KUKA KRL program: EPS_2_26056_SANMH1A_A_20260107125654.src

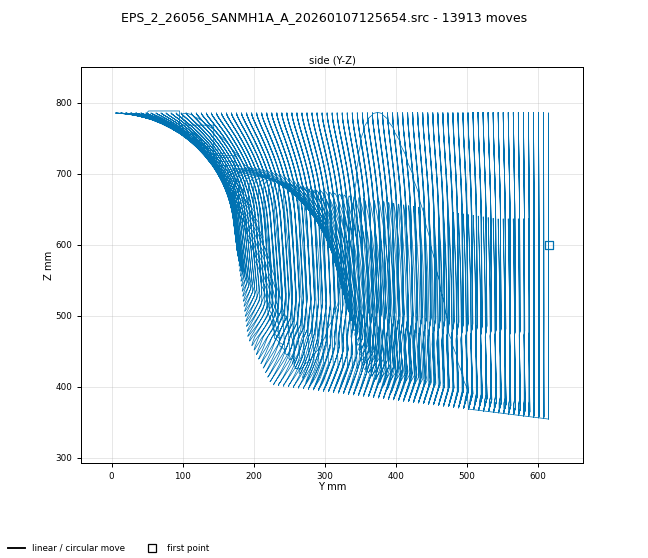
[picture p0: tool path of EPS_2_26056_SANMH1A_A_20260107125654.src, 13913 of 13915 moves have a stored position in this frame; points joined in program order, loops and branches not executed]
&ACCESS RVP
&REL 4
&COMMENT QRS 19112012
&PARAM EDITMASK = *
DEF PART()
EXT BAS (BAS_COMMAND :IN,REAL :IN )
INT I
BAS (#INITMOV,0 )

;KUKA QRS Post kuka4.cps  Date:22-06-2017 !

File_ID=2959

QRS_PRE_INIT()

;Init var - Until changes are made in qrs_pre_init
Outlet_Square_prg=0
Inlet_1_Square_prg=0
Inlet_2_Square_prg=0
Inlet_3_Square_prg=0
Inlet_4_Square_prg=0
Inlet_5_Square_prg=0

Outlet_1={X 0.000, Y 512.360, Z 637.000, B 0.000, E1 0.000 }
Inlet_1={X 0.000, Y 512.360, Z 637.000, B 0.000, E1 180.000 }
Inlet_2={X 0.000, Y 540.930, Z 321.000, B 0.000, E1 270.000 }
Outlet_1_type=299
Inlet_1_type=299
Inlet_2_type=251
;QRS#1=Sidecore dimensions
;QRS#2=300-12" PVC SDR 35
;QRS#3=300-12" PVC SDR 35
;QRS#4=250-10" PVC SDR 35
;QRS#5=
;QRS#6=
;QRS#7=
;QRS#8=
;QRS#9=16M PSX
;QRS#10=16M PSX
;QRS#11=14M PSX
;QRS#12=
;QRS#13=
;QRS#14=
;QRS#15=
;QRS#16=1220x127x1067 3,5'
;QRS#17=EPS Height
;QRS#18=786,5
;QRS#19=*
;QRS#20= UPDATED VERSION 22-06-2017
;QRS#21=*
Outlet_Square=0150
Inlet_1_Square=0150
Inlet_2_Square=0100
Inlet_3_Square=0
Inlet_4_Square=0
Inlet_5_Square=0
Mill_Square=1
Outlet_Square_Prg=206
Inlet_1_Square_prg=206
Inlet_2_Square_prg=205

QRS_INIT()

$ADVANCE=5

; T1
PTP {E1 173.596,E2 173.596}
PTP {X 0,Y 615.515,A -85,B 0,C 180,E1 173.596,E2 173.596,E3 0,E4 0,E5 0,E6 0}
QRS_SPEED_INIT()
LIN {X 0,Y 615.515,Z 600,A -85,B 0,C 180,E1 173.596,E2 173.596,E3 0,E4 0,E5 0,E6 0} C_VEL
LIN {X 0,Y 615.515,Z 364.495,A -85,B 0,C 180,E1 173.596,E2 173.596} C_VEL
LIN {X 0,Y 615.515,Z 356.328,A -85,B 0,C 180,E1 173.596,E2 173.596} C_VEL
LIN {X 0,Y 615.484,Z 354.328,A -85,B 0,C 180,E1 173.41,E2 173.41} C_VEL
LIN {X 0,Y 615.426,Z 354.324,A -85,B 0,C 180,E1 170.8,E2 170.8} C_VEL
LIN {X 0,Y 615.427,Z 354.324,A -85,B 0,C 180,E1 168.806,E2 168.806} C_VEL
LIN {X 0,Y 615.427,Z 354.324,A -85,B 0,C 180,E1 166.797,E2 166.797} C_VEL
LIN {X 0,Y 615.426,Z 354.324,A -85,B 0,C 180,E1 164.772,E2 164.772} C_VEL
LIN {X 0,Y 615.424,Z 354.324,A -85,B 0,C 180,E1 162.728,E2 162.728} C_VEL
LIN {X 0,Y 615.42,Z 354.324,A -85,B 0,C 180,E1 160.66,E2 160.66} C_VEL
LIN {X 0,Y 615.416,Z 354.324,A -85,B 0,C 180,E1 158.565,E2 158.565} C_VEL
LIN {X 0,Y 615.413,Z 354.324,A -85,B 0,C 180,E1 156.441,E2 156.441} C_VEL
LIN {X 0,Y 615.412,Z 354.324,A -85,B 0,C 180,E1 154.281,E2 154.281} C_VEL
LIN {X 0,Y 615.465,Z 354.323,A -85,B 0,C 180,E1 151.55,E2 151.55} C_VEL
LIN {X 0,Y 615.448,Z 354.325,A -85,B 0,C 180,E1 148.917,E2 148.917} C_VEL
LIN {X 0,Y 615.415,Z 354.324,A -85,B 0,C 180,E1 146.473,E2 146.473} C_VEL
LIN {X 0,Y 615.412,Z 354.324,A -85,B 0,C 180,E1 144.173,E2 144.173} C_VEL
LIN {X 0,Y 615.422,Z 354.323,A -85,B 0,C 180,E1 141.927,E2 141.927} C_VEL
LIN {X 0,Y 615.467,Z 354.326,A -85,B 0,C 180,E1 139.392,E2 139.392} C_VEL
LIN {X 0,Y 615.436,Z 354.325,A -85,B 0,C 180,E1 136.751,E2 136.751} C_VEL
LIN {X 0,Y 615.411,Z 354.324,A -85,B 0,C 180,E1 134.154,E2 134.154} C_VEL
LIN {X 0,Y 615.413,Z 354.324,A -85,B 0,C 180,E1 132.072,E2 132.072} C_VEL
LIN {X 0,Y 615.43,Z 354.323,A -85,B 0,C 180,E1 129.753,E2 129.753} C_VEL
LIN {X 0,Y 615.465,Z 354.325,A -85,B 0,C 180,E1 126.934,E2 126.934} C_VEL
LIN {X 0,Y 615.413,Z 354.324,A -85,B 0,C 180,E1 124.025,E2 124.025} C_VEL
LIN {X 0,Y 615.431,Z 354.323,A -85,B 0,C 180,E1 121.687,E2 121.687} C_VEL
LIN {X 0,Y 615.498,Z 354.495,A -85,B 0,C 180,E1 118.983,E2 118.983} C_VEL
LIN {X 0,Y 615.499,Z 355.379,A -85,B 0,C 180,E1 118.842,E2 118.842} C_VEL
LIN {X 0,Y 615.468,Z 383.107,A -85,B 0,C 180,E1 116.261,E2 116.261} C_VEL
LIN {X 0,Y 615.463,Z 411.593,A -85,B 0,C 180,E1 113.667,E2 113.667} C_VEL
LIN {X 0,Y 615.498,Z 440.574,A -85,B 0,C 180,E1 111.079,E2 111.079} C_VEL
LIN {X 0,Y 615.486,Z 472.602,A -85,B 0,C 180,E1 108.278,E2 108.278} C_VEL
LIN {X 0,Y 615.487,Z 474.74,A -85,B 0,C 180,E1 108.197,E2 108.197} C_VEL
LIN {X 0,Y 615.498,Z 640.194,A -85,B 0,C 180,E1 106.201,E2 106.201} C_VEL
LIN {X 0,Y 615.49,Z 654.874,A -85,B 0,C 180,E1 105.904,E2 105.904} C_VEL
LIN {X 0,Y 615.48,Z 669.457,A -85,B 0,C 180,E1 105.479,E2 105.479} C_VEL
LIN {X 0,Y 615.492,Z 682.768,A -85,B 0,C 180,E1 104.971,E2 104.971} C_VEL
LIN {X 0,Y 615.485,Z 696.395,A -85,B 0,C 180,E1 104.319,E2 104.319} C_VEL
LIN {X 0,Y 615.5,Z 709.685,A -85,B 0,C 180,E1 103.536,E2 103.536} C_VEL
LIN {X 0,Y 615.497,Z 721.532,A -85,B 0,C 180,E1 102.696,E2 102.696} C_VEL
LIN {X 0,Y 615.497,Z 733.373,A -85,B 0,C 180,E1 101.692,E2 101.692} C_VEL
LIN {X 0,Y 615.495,Z 743.166,A -85,B 0,C 180,E1 100.708,E2 100.708} C_VEL
LIN {X 0,Y 615.495,Z 753.021,A -85,B 0,C 180,E1 99.529,E2 99.529} C_VEL
LIN {X 0,Y 615.497,Z 761.11,A -85,B 0,C 180,E1 98.37,E2 98.37} C_VEL
LIN {X 0,Y 615.492,Z 767.789,A -85,B 0,C 180,E1 97.214,E2 97.214} C_VEL
LIN {X 0,Y 615.495,Z 773.954,A -85,B 0,C 180,E1 95.897,E2 95.897} C_VEL
LIN {X 0,Y 615.489,Z 778.72,A -85,B 0,C 180,E1 94.583,E2 94.583} C_VEL
LIN {X 0,Y 615.491,Z 782.223,A -85,B 0,C 180,E1 93.272,E2 93.272} C_VEL
LIN {X 0,Y 615.499,Z 784.541,A -85,B 0,C 180,E1 91.962,E2 91.962} C_VEL
LIN {X 0,Y 615.491,Z 785.728,A -85,B 0,C 180,E1 90.653,E2 90.653} C_VEL
LIN {X 0,Y 615.492,Z 785.751,A -85,B 0,C 180,E1 89.345,E2 89.345} C_VEL
LIN {X 0,Y 615.499,Z 784.644,A -85,B 0,C 180,E1 88.036,E2 88.036} C_VEL
LIN {X 0,Y 615.494,Z 782.413,A -85,B 0,C 180,E1 86.726,E2 86.726} C_VEL
LIN {X 0,Y 615.49,Z 779.002,A -85,B 0,C 180,E1 85.415,E2 85.415} C_VEL
LIN {X 0,Y 615.496,Z 774.332,A -85,B 0,C 180,E1 84.101,E2 84.101} C_VEL
LIN {X 0,Y 615.494,Z 768.266,A -85,B 0,C 180,E1 82.783,E2 82.783} C_VEL
LIN {X 0,Y 615.49,Z 760.627,A -85,B 0,C 180,E1 81.462,E2 81.462} C_VEL
LIN {X 0,Y 615.496,Z 752.443,A -85,B 0,C 180,E1 80.303,E2 80.303} C_VEL
LIN {X 0,Y 615.496,Z 742.329,A -85,B 0,C 180,E1 79.108,E2 79.108} C_VEL
LIN {X 0,Y 615.498,Z 730.672,A -85,B 0,C 180,E1 77.971,E2 77.971} C_VEL
LIN {X 0,Y 615.498,Z 719.4,A -85,B 0,C 180,E1 77.05,E2 77.05} C_VEL
LIN {X 0,Y 615.498,Z 707.158,A -85,B 0,C 180,E1 76.209,E2 76.209} C_VEL
LIN {X 0,Y 615.478,Z 693.757,A -85,B 0,C 180,E1 75.45,E2 75.45} C_VEL
LIN {X 0,Y 615.492,Z 679.889,A -85,B 0,C 180,E1 74.816,E2 74.816} C_VEL
LIN {X 0,Y 615.481,Z 665.667,A -85,B 0,C 180,E1 74.306,E2 74.306} C_VEL
LIN {X 0,Y 615.499,Z 651.574,A -85,B 0,C 180,E1 73.93,E2 73.93} C_VEL
LIN {X 0,Y 615.497,Z 637.157,A -85,B 0,C 180,E1 73.666,E2 73.666} C_VEL
LIN {X 0,Y 615.484,Z 473.34,A -85,B 0,C 180,E1 71.681,E2 71.681} C_VEL
LIN {X 0,Y 615.494,Z 445.533,A -85,B 0,C 180,E1 69.269,E2 69.269} C_VEL
LIN {X 0,Y 615.495,Z 415.789,A -85,B 0,C 180,E1 66.622,E2 66.622} C_VEL
LIN {X 0,Y 615.489,Z 386.043,A -85,B 0,C 180,E1 63.92,E2 63.92} C_VEL
LIN {X 0,Y 615.497,Z 356.297,A -85,B 0,C 180,E1 61.155,E2 61.155} C_VEL
LIN {X 0,Y 615.497,Z 354.615,A -85,B 0,C 180,E1 60.968,E2 60.968} C_VEL
LIN {X 0,Y 615.425,Z 354.325,A -85,B 0,C 180,E1 60.216,E2 60.216} C_VEL
LIN {X 0,Y 615.432,Z 354.325,A -85,B 0,C 180,E1 58.311,E2 58.311} C_VEL
LIN {X 0,Y 615.41,Z 354.325,A -85,B 0,C 180,E1 55.972,E2 55.972} C_VEL
LIN {X 0,Y 615.46,Z 354.325,A -85,B 0,C 180,E1 53.067,E2 53.067} C_VEL
LIN {X 0,Y 615.429,Z 354.324,A -85,B 0,C 180,E1 50.245,E2 50.245} C_VEL
LIN {X 0,Y 615.414,Z 354.324,A -85,B 0,C 180,E1 47.928,E2 47.928} C_VEL
LIN {X 0,Y 615.413,Z 354.324,A -85,B 0,C 180,E1 45.843,E2 45.843} C_VEL
LIN {X 0,Y 615.442,Z 354.324,A -85,B 0,C 180,E1 43.249,E2 43.249} C_VEL
LIN {X 0,Y 615.47,Z 354.323,A -85,B 0,C 180,E1 40.608,E2 40.608} C_VEL
LIN {X 0,Y 615.423,Z 354.322,A -85,B 0,C 180,E1 38.004,E2 38.004} C_VEL
LIN {X 0,Y 615.422,Z 354.323,A -85,B 0,C 180,E1 35.62,E2 35.62} C_VEL
LIN {X 0,Y 615.448,Z 354.324,A -85,B 0,C 180,E1 33.239,E2 33.239} C_VEL
LIN {X 0,Y 615.489,Z 354.325,A -85,B 0,C 180,E1 30.92,E2 30.92} C_VEL
LIN {X 0,Y 615.468,Z 354.319,A -85,B 0,C 180,E1 28.446,E2 28.446} C_VEL
LIN {X 0,Y 615.468,Z 354.318,A -85,B 0,C 180,E1 26.445,E2 26.445} C_VEL
LIN {X 0,Y 615.433,Z 354.32,A -85,B 0,C 180,E1 23.996,E2 23.996} C_VEL
LIN {X 0,Y 615.443,Z 354.319,A -85,B 0,C 180,E1 22.138,E2 22.138} C_VEL
LIN {X 0,Y 615.437,Z 354.319,A -85,B 0,C 180,E1 20.035,E2 20.035} C_VEL
LIN {X 0,Y 615.498,Z 354.519,A -85,B 0,C 180,E1 18.797,E2 18.797} C_VEL
LIN {X 0,Y 615.492,Z 371.153,A -85,B 0,C 180,E1 16.167,E2 16.167} C_VEL
LIN {X 0,Y 615.457,Z 375.25,A -85,B 0,C 180,E1 15.566,E2 15.566} C_VEL
LIN {X 0,Y 615.454,Z 377.392,A -85,B 0,C 180,E1 15.503,E2 15.503} C_VEL
LIN {X 0,Y 615.498,Z 511.173,A -85,B 0,C 180,E1 13.905,E2 13.905} C_VEL
LIN {X 0,Y 615.497,Z 524.744,A -85,B 0,C 180,E1 13.621,E2 13.621} C_VEL
LIN {X 0,Y 615.497,Z 538.485,A -85,B 0,C 180,E1 13.201,E2 13.201} C_VEL
LIN {X 0,Y 615.493,Z 550.898,A -85,B 0,C 180,E1 12.698,E2 12.698} C_VEL
LIN {X 0,Y 615.486,Z 563.841,A -85,B 0,C 180,E1 12.028,E2 12.028} C_VEL
LIN {X 0,Y 615.499,Z 575.557,A -85,B 0,C 180,E1 11.276,E2 11.276} C_VEL
LIN {X 0,Y 615.498,Z 587.225,A -85,B 0,C 180,E1 10.36,E2 10.36} C_VEL
LIN {X 0,Y 615.497,Z 597.649,A -85,B 0,C 180,E1 9.364,E2 9.364} C_VEL
LIN {X 0,Y 615.496,Z 606.239,A -85,B 0,C 180,E1 8.371,E2 8.371} C_VEL
LIN {X 0,Y 615.495,Z 614.452,A -85,B 0,C 180,E1 7.216,E2 7.216} C_VEL
LIN {X 0,Y 615.496,Z 620.183,A -85,B 0,C 180,E1 6.227,E2 6.227} C_VEL
LIN {X 0,Y 615.495,Z 624.887,A -85,B 0,C 180,E1 5.241,E2 5.241} C_VEL
LIN {X 0,Y 615.494,Z 629.757,A -85,B 0,C 180,E1 3.929,E2 3.929} C_VEL
LIN {X 0,Y 615.496,Z 633.154,A -85,B 0,C 180,E1 2.618,E2 2.618} C_VEL
LIN {X 0,Y 615.494,Z 635.174,A -85,B 0,C 180,E1 1.309,E2 1.309} C_VEL
LIN {X 0,Y 615.491,Z 635.885,A -85,B 0,C 180,E1 0,E2 0} C_VEL
LIN {X 0,Y 615.489,Z 635.28,A -85,B 0,C 180,E1 -1.309,E2 -1.309} C_VEL
LIN {X 0,Y 615.497,Z 633.35,A -85,B 0,C 180,E1 -2.618,E2 -2.618} C_VEL
LIN {X 0,Y 615.494,Z 630.046,A -85,B 0,C 180,E1 -3.928,E2 -3.928} C_VEL
LIN {X 0,Y 615.495,Z 625.274,A -85,B 0,C 180,E1 -5.241,E2 -5.241} C_VEL
LIN {X 0,Y 615.497,Z 618.874,A -85,B 0,C 180,E1 -6.557,E2 -6.557} C_VEL
LIN {X 0,Y 615.496,Z 611.744,A -85,B 0,C 180,E1 -7.71,E2 -7.71} C_VEL
LIN {X 0,Y 615.498,Z 604.271,A -85,B 0,C 180,E1 -8.702,E2 -8.702} C_VEL
LIN {X 0,Y 615.495,Z 595.292,A -85,B 0,C 180,E1 -9.696,E2 -9.696} C_VEL
LIN {X 0,Y 615.498,Z 584.208,A -85,B 0,C 180,E1 -10.709,E2 -10.709} C_VEL
LIN {X 0,Y 615.498,Z 573.281,A -85,B 0,C 180,E1 -11.526,E2 -11.526} C_VEL
LIN {X 0,Y 615.486,Z 560.984,A -85,B 0,C 180,E1 -12.279,E2 -12.279} C_VEL
LIN {X 0,Y 615.488,Z 549.146,A -85,B 0,C 180,E1 -12.865,E2 -12.865} C_VEL
LIN {X 0,Y 615.494,Z 536.22,A -85,B 0,C 180,E1 -13.369,E2 -13.369} C_VEL
LIN {X 0,Y 615.498,Z 523.24,A -85,B 0,C 180,E1 -13.748,E2 -13.748} C_VEL
LIN {X 0,Y 615.497,Z 510.029,A -85,B 0,C 180,E1 -14.012,E2 -14.012} C_VEL
LIN {X 0,Y 615.491,Z 375.663,A -85,B 0,C 180,E1 -15.629,E2 -15.629} C_VEL
LIN {X 0,Y 615.495,Z 374.551,A -85,B 0,C 180,E1 -15.735,E2 -15.735} C_VEL
LIN {X 0,Y 615.496,Z 355.917,A -85,B 0,C 180,E1 -18.646,E2 -18.646} C_VEL
LIN {X 0,Y 615.496,Z 354.46,A -85,B 0,C 180,E1 -18.905,E2 -18.905} C_VEL
LIN {X 0,Y 615.491,Z 354.311,A -85,B 0,C 180,E1 -21.432,E2 -21.432} C_VEL
LIN {X 0,Y 615.469,Z 354.316,A -85,B 0,C 180,E1 -24.273,E2 -24.273} C_VEL
LIN {X 0,Y 615.481,Z 354.319,A -85,B 0,C 180,E1 -27.043,E2 -27.043} C_VEL
LIN {X 0,Y 615.488,Z 354.308,A -85,B 0,C 180,E1 -29.794,E2 -29.794} C_VEL
LIN {X 0,Y 615.487,Z 354.323,A -85,B 0,C 180,E1 -32.457,E2 -32.457} C_VEL
LIN {X 0,Y 615.476,Z 354.32,A -85,B 0,C 180,E1 -34.816,E2 -34.816} C_VEL
LIN {X 0,Y 615.467,Z 354.314,A -85,B 0,C 180,E1 -37.244,E2 -37.244} C_VEL
LIN {X 0,Y 615.489,Z 354.318,A -85,B 0,C 180,E1 -40.088,E2 -40.088} C_VEL
LIN {X 0,Y 615.494,Z 354.325,A -85,B 0,C 180,E1 -42.352,E2 -42.352} C_VEL
LIN {X 0,Y 615.448,Z 354.317,A -85,B 0,C 180,E1 -45.072,E2 -45.072} C_VEL
LIN {X 0,Y 615.497,Z 354.318,A -85,B 0,C 180,E1 -47.919,E2 -47.919} C_VEL
LIN {X 0,Y 615.475,Z 354.325,A -85,B 0,C 180,E1 -50.248,E2 -50.248} C_VEL
LIN {X 0,Y 615.43,Z 354.322,A -85,B 0,C 180,E1 -52.753,E2 -52.753} C_VEL
LIN {X 0,Y 615.438,Z 354.322,A -85,B 0,C 180,E1 -55.306,E2 -55.306} C_VEL
LIN {X 0,Y 615.438,Z 354.325,A -85,B 0,C 180,E1 -58.311,E2 -58.311} C_VEL
LIN {X 0,Y 615.416,Z 354.325,A -85,B 0,C 180,E1 -60.589,E2 -60.589} C_VEL
LIN {X 0,Y 615.496,Z 354.507,A -85,B 0,C 180,E1 -61.886,E2 -61.886} C_VEL
LIN {X 0,Y 615.494,Z 355.377,A -85,B 0,C 180,E1 -62.018,E2 -62.018} C_VEL
LIN {X 0,Y 615.482,Z 387.128,A -85,B 0,C 180,E1 -64.721,E2 -64.721} C_VEL
LIN {X 0,Y 615.499,Z 419.368,A -85,B 0,C 180,E1 -67.404,E2 -67.404} C_VEL
LIN {X 0,Y 615.479,Z 452.912,A -85,B 0,C 180,E1 -70.14,E2 -70.14} C_VEL
LIN {X 0,Y 615.486,Z 472.762,A -85,B 0,C 180,E1 -71.72,E2 -71.72} C_VEL
LIN {X 0,Y 615.498,Z 640.913,A -85,B 0,C 180,E1 -73.764,E2 -73.764} C_VEL
LIN {X 0,Y 615.49,Z 656.681,A -85,B 0,C 180,E1 -74.094,E2 -74.094} C_VEL
LIN {X 0,Y 615.48,Z 672.028,A -85,B 0,C 180,E1 -74.561,E2 -74.561} C_VEL
LIN {X 0,Y 615.484,Z 685.734,A -85,B 0,C 180,E1 -75.112,E2 -75.112} C_VEL
LIN {X 0,Y 615.493,Z 700.041,A -85,B 0,C 180,E1 -75.833,E2 -75.833} C_VEL
LIN {X 0,Y 615.497,Z 712.886,A -85,B 0,C 180,E1 -76.63,E2 -76.63} C_VEL
LIN {X 0,Y 615.495,Z 725.244,A -85,B 0,C 180,E1 -77.553,E2 -77.553} C_VEL
LIN {X 0,Y 615.495,Z 735.597,A -85,B 0,C 180,E1 -78.473,E2 -78.473} C_VEL
LIN {X 0,Y 615.494,Z 745.176,A -85,B 0,C 180,E1 -79.472,E2 -79.472} C_VEL
LIN {X 0,Y 615.495,Z 754.57,A -85,B 0,C 180,E1 -80.635,E2 -80.635} C_VEL
LIN {X 0,Y 615.496,Z 762.375,A -85,B 0,C 180,E1 -81.793,E2 -81.793} C_VEL
LIN {X 0,Y 615.497,Z 769.605,A -85,B 0,C 180,E1 -83.102,E2 -83.102} C_VEL
LIN {X 0,Y 615.499,Z 775.433,A -85,B 0,C 180,E1 -84.429,E2 -84.429} C_VEL
LIN {X 0,Y 615.491,Z 778.857,A -85,B 0,C 180,E1 -85.415,E2 -85.415} C_VEL
LIN {X 0,Y 615.492,Z 782.316,A -85,B 0,C 180,E1 -86.726,E2 -86.726} C_VEL
LIN {X 0,Y 615.496,Z 784.592,A -85,B 0,C 180,E1 -88.036,E2 -88.036} C_VEL
LIN {X 0,Y 615.493,Z 785.74,A -85,B 0,C 180,E1 -89.345,E2 -89.345} C_VEL
LIN {X 0,Y 615.493,Z 785.741,A -85,B 0,C 180,E1 -90.653,E2 -90.653} C_VEL
LIN {X 0,Y 615.495,Z 784.595,A -85,B 0,C 180,E1 -91.962,E2 -91.962} C_VEL
LIN {X 0,Y 615.492,Z 782.32,A -85,B 0,C 180,E1 -93.272,E2 -93.272} C_VEL
LIN {X 0,Y 615.491,Z 778.864,A -85,B 0,C 180,E1 -94.583,E2 -94.583} C_VEL
LIN {X 0,Y 615.49,Z 774.148,A -85,B 0,C 180,E1 -95.897,E2 -95.897} C_VEL
LIN {X 0,Y 615.496,Z 768.035,A -85,B 0,C 180,E1 -97.214,E2 -97.214} C_VEL
LIN {X 0,Y 615.49,Z 760.341,A -85,B 0,C 180,E1 -98.535,E2 -98.535} C_VEL
LIN {X 0,Y 615.495,Z 752.122,A -85,B 0,C 180,E1 -99.695,E2 -99.695} C_VEL
LIN {X 0,Y 615.496,Z 741.897,A -85,B 0,C 180,E1 -100.892,E2 -100.892} C_VEL
LIN {X 0,Y 615.495,Z 732.08,A -85,B 0,C 180,E1 -101.859,E2 -101.859} C_VEL
LIN {X 0,Y 615.497,Z 719.964,A -85,B 0,C 180,E1 -102.864,E2 -102.864} C_VEL
LIN {X 0,Y 615.498,Z 707.816,A -85,B 0,C 180,E1 -103.704,E2 -103.704} C_VEL
LIN {X 0,Y 615.477,Z 694.399,A -85,B 0,C 180,E1 -104.472,E2 -104.472} C_VEL
LIN {X 0,Y 615.495,Z 679.877,A -85,B 0,C 180,E1 -105.14,E2 -105.14} C_VEL
LIN {X 0,Y 615.48,Z 665.654,A -85,B 0,C 180,E1 -105.649,E2 -105.649} C_VEL
LIN {X 0,Y 615.5,Z 651.125,A -85,B 0,C 180,E1 -106.036,E2 -106.036} C_VEL
LIN {X 0,Y 615.498,Z 636.349,A -85,B 0,C 180,E1 -106.301,E2 -106.301} C_VEL
LIN {X 0,Y 615.487,Z 472.791,A -85,B 0,C 180,E1 -108.279,E2 -108.279} C_VEL
LIN {X 0,Y 615.481,Z 441.108,A -85,B 0,C 180,E1 -110.817,E2 -110.817} C_VEL
LIN {X 0,Y 615.487,Z 407.768,A -85,B 0,C 180,E1 -113.555,E2 -113.555} C_VEL
LIN {X 0,Y 615.496,Z 374.428,A -85,B 0,C 180,E1 -116.351,E2 -116.351} C_VEL
LIN {X 0,Y 615.495,Z 354.685,A -85,B 0,C 180,E1 -118.062,E2 -118.062} C_VEL
LIN {X 0,Y 615.464,Z 354.326,A -85,B 0,C 180,E1 -118.446,E2 -118.446} C_VEL
LIN {X 0,Y 615.422,Z 354.324,A -85,B 0,C 180,E1 -120.922,E2 -120.922} C_VEL
LIN {X 0,Y 615.414,Z 354.323,A -85,B 0,C 180,E1 -123.239,E2 -123.239} C_VEL
LIN {X 0,Y 615.447,Z 354.322,A -85,B 0,C 180,E1 -125.828,E2 -125.828} C_VEL
LIN {X 0,Y 615.477,Z 354.322,A -85,B 0,C 180,E1 -128.067,E2 -128.067} C_VEL
LIN {X 0,Y 615.455,Z 354.324,A -85,B 0,C 180,E1 -130.607,E2 -130.607} C_VEL
LIN {X 0,Y 615.419,Z 354.324,A -85,B 0,C 180,E1 -133.041,E2 -133.041} C_VEL
LIN {X 0,Y 615.418,Z 354.324,A -85,B 0,C 180,E1 -135.073,E2 -135.073} C_VEL
LIN {X 0,Y 615.421,Z 354.324,A -85,B 0,C 180,E1 -137.641,E2 -137.641} C_VEL
LIN {X 0,Y 615.496,Z 354.322,A -85,B 0,C 180,E1 -140.251,E2 -140.251} C_VEL
LIN {X 0,Y 615.42,Z 354.324,A -85,B 0,C 180,E1 -143.069,E2 -143.069} C_VEL
LIN {X 0,Y 615.411,Z 354.324,A -85,B 0,C 180,E1 -145.307,E2 -145.307} C_VEL
LIN {X 0,Y 615.416,Z 354.323,A -85,B 0,C 180,E1 -147.538,E2 -147.538} C_VEL
LIN {X 0,Y 615.476,Z 354.323,A -85,B 0,C 180,E1 -150.204,E2 -150.204} C_VEL
LIN {X 0,Y 615.429,Z 354.324,A -85,B 0,C 180,E1 -152.962,E2 -152.962} C_VEL
LIN {X 0,Y 615.428,Z 354.324,A -85,B 0,C 180,E1 -155.006,E2 -155.006} C_VEL
LIN {X 0,Y 615.419,Z 354.324,A -85,B 0,C 180,E1 -157.153,E2 -157.153} C_VEL
LIN {X 0,Y 615.413,Z 354.323,A -85,B 0,C 180,E1 -159.457,E2 -159.457} C_VEL
LIN {X 0,Y 615.448,Z 354.323,A -85,B 0,C 180,E1 -162.042,E2 -162.042} C_VEL
LIN {X 0,Y 615.456,Z 354.325,A -85,B 0,C 180,E1 -164.773,E2 -164.773} C_VEL
LIN {X 0,Y 615.413,Z 354.324,A -85,B 0,C 180,E1 -167.468,E2 -167.468} C_VEL
LIN {X 0,Y 615.45,Z 354.323,A -85,B 0,C 180,E1 -170.137,E2 -170.137} C_VEL
LIN {X 0,Y 615.46,Z 354.325,A -85,B 0,C 180,E1 -172.784,E2 -172.784} C_VEL
LIN {X 0,Y 615.413,Z 354.324,A -85,B 0,C 180,E1 -175.415,E2 -175.415} C_VEL
LIN {X 0,Y 615.412,Z 354.324,A -85,B 0,C 180,E1 -177.382,E2 -177.382} C_VEL
LIN {X 0,Y 615.416,Z 354.324,A -85,B 0,C 180,E1 -179.346,E2 -179.346} C_VEL
LIN {X 0,Y 615.418,Z 354.324,A -85,B 0,C 180,E1 -181.309,E2 -181.309} C_VEL
LIN {X 0,Y 615.417,Z 354.325,A -85,B 0,C 180,E1 -183.273,E2 -183.273} C_VEL
LIN {X 0,Y 615.421,Z 354.324,A -85,B 0,C 180,E1 -185.242,E2 -185.242} C_VEL
LIN {X 0,Y 615.484,Z 354.328,A -85,B 0,C 180,E1 -186.59,E2 -186.59} C_VEL
LIN {X 0,Y 614.769,Z 354.468,A -85,B 0,C 180,E1 -187.136,E2 -187.136} C_VEL
LIN {X 0,Y 611.909,Z 354.883,A -85,B 0,C 180,E1 -188.022,E2 -188.022} C_VEL
LIN {X 0,Y 609.519,Z 355.192,A -85,B 0,C 180,E1 -188.734,E2 -188.734} C_VEL
LIN {X 0,Y 608.49,Z 355.309,A -85,B 0,C 180,E1 -189.284,E2 -189.284} C_VEL
LIN {X 0,Y 608.402,Z 355.318,A -85,B 0,C 180,E1 -189.47,E2 -189.47} C_VEL
LIN {X 0,Y 608.414,Z 355.318,A -85,B 0,C 180,E1 -192.001,E2 -192.001} C_VEL
LIN {X 0,Y 608.454,Z 355.321,A -85,B 0,C 180,E1 -194.721,E2 -194.721} C_VEL
LIN {X 0,Y 608.394,Z 355.319,A -85,B 0,C 180,E1 -197.478,E2 -197.478} C_VEL
LIN {X 0,Y 608.393,Z 355.319,A -85,B 0,C 180,E1 -199.573,E2 -199.573} C_VEL
LIN {X 0,Y 608.41,Z 355.317,A -85,B 0,C 180,E1 -201.694,E2 -201.694} C_VEL
LIN {X 0,Y 608.421,Z 355.325,A -85,B 0,C 180,E1 -204.573,E2 -204.573} C_VEL
LIN {X 0,Y 608.399,Z 355.319,A -85,B 0,C 180,E1 -207.521,E2 -207.521} C_VEL
LIN {X 0,Y 608.399,Z 355.318,A -85,B 0,C 180,E1 -209.783,E2 -209.783} C_VEL
LIN {X 0,Y 608.44,Z 355.321,A -85,B 0,C 180,E1 -212.522,E2 -212.522} C_VEL
LIN {X 0,Y 608.404,Z 355.321,A -85,B 0,C 180,E1 -215.28,E2 -215.28} C_VEL
LIN {X 0,Y 608.391,Z 355.319,A -85,B 0,C 180,E1 -217.752,E2 -217.752} C_VEL
LIN {X 0,Y 608.42,Z 355.319,A -85,B 0,C 180,E1 -220.328,E2 -220.328} C_VEL
LIN {X 0,Y 608.428,Z 355.318,A -85,B 0,C 180,E1 -223.307,E2 -223.307} C_VEL
LIN {X 0,Y 608.415,Z 355.318,A -85,B 0,C 180,E1 -226.128,E2 -226.128} C_VEL
LIN {X 0,Y 608.439,Z 355.325,A -85,B 0,C 180,E1 -228.824,E2 -228.824} C_VEL
LIN {X 0,Y 608.398,Z 355.321,A -85,B 0,C 180,E1 -231.409,E2 -231.409} C_VEL
LIN {X 0,Y 608.433,Z 355.321,A -85,B 0,C 180,E1 -233.085,E2 -233.085} C_VEL
LIN {X 0,Y 608.418,Z 355.317,A -85,B 0,C 180,E1 -235.529,E2 -235.529} C_VEL
LIN {X 0,Y 608.405,Z 355.318,A -85,B 0,C 180,E1 -237.904,E2 -237.904} C_VEL
LIN {X 0,Y 608.484,Z 355.462,A -85,B 0,C 180,E1 -240.769,E2 -240.769} C_VEL
LIN {X 0,Y 608.894,Z 357.354,A -85,B 0,C 180,E1 -241.004,E2 -241.004} C_VEL
LIN {X 0,Y 608.778,Z 385.095,A -85,B 0,C 180,E1 -243.613,E2 -243.613} C_VEL
LIN {X 0,Y 608.705,Z 412.837,A -85,B 0,C 180,E1 -246.166,E2 -246.166} C_VEL
LIN {X 0,Y 608.666,Z 442.562,A -85,B 0,C 180,E1 -248.85,E2 -248.85} C_VEL
LIN {X 0,Y 608.623,Z 473.186,A -85,B 0,C 180,E1 -251.549,E2 -251.549} C_VEL
LIN {X 0,Y 608.762,Z 478.084,A -85,B 0,C 180,E1 -251.635,E2 -251.635} C_VEL
LIN {X 0,Y 608.698,Z 641.301,A -85,B 0,C 180,E1 -253.629,E2 -253.629} C_VEL
LIN {X 0,Y 608.648,Z 656.678,A -85,B 0,C 180,E1 -253.956,E2 -253.956} C_VEL
LIN {X 0,Y 608.64,Z 672.026,A -85,B 0,C 180,E1 -254.428,E2 -254.428} C_VEL
LIN {X 0,Y 608.591,Z 686.699,A -85,B 0,C 180,E1 -255.027,E2 -255.027} C_VEL
LIN {X 0,Y 608.571,Z 700.458,A -85,B 0,C 180,E1 -255.736,E2 -255.736} C_VEL
LIN {X 0,Y 608.547,Z 713.56,A -85,B 0,C 180,E1 -256.562,E2 -256.562} C_VEL
LIN {X 0,Y 608.505,Z 725.854,A -85,B 0,C 180,E1 -257.494,E2 -257.494} C_VEL
LIN {X 0,Y 608.497,Z 737.061,A -85,B 0,C 180,E1 -258.509,E2 -258.509} C_VEL
LIN {X 0,Y 608.477,Z 747.946,A -85,B 0,C 180,E1 -259.688,E2 -259.688} C_VEL
LIN {X 0,Y 608.469,Z 756.992,A -85,B 0,C 180,E1 -260.863,E2 -260.863} C_VEL
LIN {X 0,Y 608.459,Z 764.487,A -85,B 0,C 180,E1 -262.034,E2 -262.034} C_VEL
LIN {X 0,Y 608.444,Z 771.634,A -85,B 0,C 180,E1 -263.398,E2 -263.398} C_VEL
LIN {X 0,Y 608.435,Z 776.998,A -85,B 0,C 180,E1 -264.699,E2 -264.699} C_VEL
LIN {X 0,Y 608.432,Z 781.17,A -85,B 0,C 180,E1 -266.027,E2 -266.027} C_VEL
LIN {X 0,Y 608.421,Z 784.111,A -85,B 0,C 180,E1 -267.353,E2 -267.353} C_VEL
LIN {X 0,Y 608.444,Z 785.881,A -85,B 0,C 180,E1 -268.677,E2 -268.677} C_VEL
LIN {X 0,Y 608.432,Z 786.496,A -85,B 0,C 180,E1 -270.001,E2 -270.001} C_VEL
LIN {X 0,Y 608.447,Z 785.943,A -85,B 0,C 180,E1 -271.325,E2 -271.325} C_VEL
LIN {X 0,Y 608.424,Z 784.258,A -85,B 0,C 180,E1 -272.649,E2 -272.649} C_VEL
LIN {X 0,Y 608.433,Z 781.405,A -85,B 0,C 180,E1 -273.975,E2 -273.975} C_VEL
LIN {X 0,Y 608.435,Z 777.325,A -85,B 0,C 180,E1 -275.303,E2 -275.303} C_VEL
LIN {X 0,Y 608.447,Z 771.917,A -85,B 0,C 180,E1 -276.634,E2 -276.634} C_VEL
LIN {X 0,Y 608.459,Z 765.017,A -85,B 0,C 180,E1 -277.968,E2 -277.968} C_VEL
LIN {X 0,Y 608.466,Z 757.586,A -85,B 0,C 180,E1 -279.139,E2 -279.139} C_VEL
LIN {X 0,Y 608.477,Z 748.657,A -85,B 0,C 180,E1 -280.314,E2 -280.314} C_VEL
LIN {X 0,Y 608.497,Z 737.94,A -85,B 0,C 180,E1 -281.493,E2 -281.493} C_VEL
LIN {X 0,Y 608.513,Z 725.892,A -85,B 0,C 180,E1 -282.592,E2 -282.592} C_VEL
LIN {X 0,Y 608.543,Z 713.602,A -85,B 0,C 180,E1 -283.526,E2 -283.526} C_VEL
LIN {X 0,Y 608.586,Z 700.655,A -85,B 0,C 180,E1 -284.343,E2 -284.343} C_VEL
LIN {X 0,Y 608.587,Z 686.749,A -85,B 0,C 180,E1 -285.061,E2 -285.061} C_VEL
LIN {X 0,Y 608.632,Z 672.081,A -85,B 0,C 180,E1 -285.66,E2 -285.66} C_VEL
LIN {X 0,Y 608.67,Z 656.473,A -85,B 0,C 180,E1 -286.139,E2 -286.139} C_VEL
LIN {X 0,Y 608.683,Z 641.356,A -85,B 0,C 180,E1 -286.46,E2 -286.46} C_VEL
LIN {X 0,Y 608.645,Z 473.638,A -85,B 0,C 180,E1 -288.522,E2 -288.522} C_VEL
LIN {X 0,Y 608.61,Z 469.321,A -85,B 0,C 180,E1 -288.865,E2 -288.865} C_VEL
LIN {X 0,Y 608.656,Z 439.578,A -85,B 0,C 180,E1 -291.507,E2 -291.507} C_VEL
LIN {X 0,Y 608.762,Z 407.768,A -85,B 0,C 180,E1 -294.384,E2 -294.384} C_VEL
LIN {X 0,Y 608.825,Z 376.586,A -85,B 0,C 180,E1 -297.27,E2 -297.27} C_VEL
LIN {X 0,Y 608.898,Z 358.273,A -85,B 0,C 180,E1 -298.998,E2 -298.998} C_VEL
LIN {X 0,Y 608.497,Z 355.53,A -85,B 0,C 180,E1 -299.303,E2 -299.303} C_VEL
LIN {X 0,Y 608.404,Z 355.319,A -85,B 0,C 180,E1 -302.099,E2 -302.099} C_VEL
LIN {X 0,Y 608.409,Z 355.323,A -85,B 0,C 180,E1 -304.9,E2 -304.9} C_VEL
LIN {X 0,Y 608.403,Z 355.321,A -85,B 0,C 180,E1 -307.752,E2 -307.752} C_VEL
LIN {X 0,Y 608.405,Z 355.318,A -85,B 0,C 180,E1 -310.324,E2 -310.324} C_VEL
LIN {X 0,Y 608.481,Z 355.317,A -85,B 0,C 180,E1 -313.31,E2 -313.31} C_VEL
LIN {X 0,Y 608.413,Z 355.317,A -85,B 0,C 180,E1 -316.125,E2 -316.125} C_VEL
LIN {X 0,Y 608.421,Z 355.321,A -85,B 0,C 180,E1 -318.821,E2 -318.821} C_VEL
LIN {X 0,Y 608.398,Z 355.321,A -85,B 0,C 180,E1 -321.769,E2 -321.769} C_VEL
LIN {X 0,Y 608.408,Z 355.318,A -85,B 0,C 180,E1 -323.96,E2 -323.96} C_VEL
LIN {X 0,Y 608.413,Z 355.317,A -85,B 0,C 180,E1 -326.326,E2 -326.326} C_VEL
LIN {X 0,Y 608.438,Z 355.318,A -85,B 0,C 180,E1 -328.735,E2 -328.735} C_VEL
LIN {X 0,Y 608.42,Z 355.318,A -85,B 0,C 180,E1 -331.732,E2 -331.732} C_VEL
LIN {X 0,Y 608.424,Z 355.316,A -85,B 0,C 180,E1 -334.289,E2 -334.289} C_VEL
LIN {X 0,Y 608.432,Z 355.321,A -85,B 0,C 180,E1 -336.875,E2 -336.875} C_VEL
LIN {X 0,Y 608.438,Z 355.316,A -85,B 0,C 180,E1 -339.725,E2 -339.725} C_VEL
LIN {X 0,Y 608.493,Z 355.5,A -85,B 0,C 180,E1 -341.132,E2 -341.132} C_VEL
LIN {X 0,Y 608.506,Z 371.897,A -85,B 0,C 180,E1 -343.743,E2 -343.743} C_VEL
LIN {X 0,Y 608.489,Z 375.574,A -85,B 0,C 180,E1 -344.272,E2 -344.272} C_VEL
LIN {X 0,Y 608.616,Z 379.226,A -85,B 0,C 180,E1 -344.34,E2 -344.34} C_VEL
LIN {X 0,Y 608.613,Z 511.923,A -85,B 0,C 180,E1 -345.947,E2 -345.947} C_VEL
LIN {X 0,Y 608.613,Z 526.305,A -85,B 0,C 180,E1 -346.264,E2 -346.264} C_VEL
LIN {X 0,Y 608.586,Z 539.65,A -85,B 0,C 180,E1 -346.689,E2 -346.689} C_VEL
LIN {X 0,Y 608.541,Z 552.707,A -85,B 0,C 180,E1 -347.24,E2 -347.24} C_VEL
LIN {X 0,Y 608.529,Z 565.343,A -85,B 0,C 180,E1 -347.917,E2 -347.917} C_VEL
LIN {X 0,Y 608.5,Z 576.851,A -85,B 0,C 180,E1 -348.677,E2 -348.677} C_VEL
LIN {X 0,Y 608.495,Z 587.412,A -85,B 0,C 180,E1 -349.519,E2 -349.519} C_VEL
LIN {X 0,Y 608.481,Z 597.898,A -85,B 0,C 180,E1 -350.527,E2 -350.527} C_VEL
LIN {X 0,Y 608.463,Z 606.55,A -85,B 0,C 180,E1 -351.531,E2 -351.531} C_VEL
LIN {X 0,Y 608.461,Z 614.837,A -85,B 0,C 180,E1 -352.7,E2 -352.7} C_VEL
LIN {X 0,Y 608.443,Z 621.325,A -85,B 0,C 180,E1 -353.832,E2 -353.832} C_VEL
LIN {X 0,Y 608.435,Z 626.787,A -85,B 0,C 180,E1 -355.03,E2 -355.03} C_VEL
LIN {X 0,Y 608.432,Z 630.298,A -85,B 0,C 180,E1 -356.026,E2 -356.026} C_VEL
LIN {X 0,Y 608.425,Z 633.734,A -85,B 0,C 180,E1 -357.352,E2 -357.352} C_VEL
LIN {X 0,Y 608.446,Z 635.777,A -85,B 0,C 180,E1 -358.676,E2 -358.676} C_VEL
LIN {X 0,Y 608.431,Z 636.495,A -85,B 0,C 180,E1 -360,E2 -360} C_VEL
LIN {X 0,Y 608.442,Z 635.882,A -85,B 0,C 180,E1 -361.324,E2 -361.324} C_VEL
LIN {X 0,Y 608.425,Z 633.929,A -85,B 0,C 180,E1 -362.648,E2 -362.648} C_VEL
LIN {X 0,Y 608.432,Z 630.586,A -85,B 0,C 180,E1 -363.974,E2 -363.974} C_VEL
LIN {X 0,Y 608.439,Z 625.761,A -85,B 0,C 180,E1 -365.302,E2 -365.302} C_VEL
LIN {X 0,Y 608.447,Z 619.458,A -85,B 0,C 180,E1 -366.603,E2 -366.603} C_VEL
LIN {X 0,Y 608.453,Z 612.102,A -85,B 0,C 180,E1 -367.8,E2 -367.8} C_VEL
LIN {X 0,Y 608.472,Z 603.203,A -85,B 0,C 180,E1 -368.971,E2 -368.971} C_VEL
LIN {X 0,Y 608.472,Z 593.867,A -85,B 0,C 180,E1 -369.977,E2 -369.977} C_VEL
LIN {X 0,Y 608.507,Z 582.624,A -85,B 0,C 180,E1 -370.972,E2 -370.972} C_VEL
LIN {X 0,Y 608.532,Z 570.832,A -85,B 0,C 180,E1 -371.829,E2 -371.829} C_VEL
LIN {X 0,Y 608.526,Z 557.912,A -85,B 0,C 180,E1 -372.591,E2 -372.591} C_VEL
LIN {X 0,Y 608.567,Z 544.232,A -85,B 0,C 180,E1 -373.227,E2 -373.227} C_VEL
LIN {X 0,Y 608.605,Z 530.273,A -85,B 0,C 180,E1 -373.715,E2 -373.715} C_VEL
LIN {X 0,Y 608.61,Z 515.882,A -85,B 0,C 180,E1 -374.069,E2 -374.069} C_VEL
LIN {X 0,Y 608.637,Z 499.023,A -85,B 0,C 180,E1 -374.316,E2 -374.316} C_VEL
LIN {X 0,Y 608.565,Z 375.878,A -85,B 0,C 180,E1 -375.801,E2 -375.801} C_VEL
LIN {X 0,Y 608.499,Z 374.625,A -85,B 0,C 180,E1 -375.921,E2 -375.921} C_VEL
LIN {X 0,Y 608.516,Z 355.97,A -85,B 0,C 180,E1 -378.868,E2 -378.868} C_VEL
LIN {X 0,Y 608.463,Z 355.362,A -85,B 0,C 180,E1 -379.044,E2 -379.044} C_VEL
LIN {X 0,Y 608.464,Z 355.312,A -85,B 0,C 180,E1 -381.692,E2 -381.692} C_VEL
LIN {X 0,Y 608.447,Z 355.32,A -85,B 0,C 180,E1 -384.571,E2 -384.571} C_VEL
LIN {X 0,Y 608.475,Z 355.313,A -85,B 0,C 180,E1 -387.206,E2 -387.206} C_VEL
LIN {X 0,Y 608.467,Z 355.312,A -85,B 0,C 180,E1 -389.971,E2 -389.971} C_VEL
LIN {X 0,Y 608.451,Z 355.318,A -85,B 0,C 180,E1 -392.88,E2 -392.88} C_VEL
LIN {X 0,Y 608.443,Z 355.314,A -85,B 0,C 180,E1 -395.278,E2 -395.278} C_VEL
LIN {X 0,Y 608.467,Z 355.318,A -85,B 0,C 180,E1 -398.239,E2 -398.239} C_VEL
LIN {X 0,Y 608.43,Z 355.316,A -85,B 0,C 180,E1 -401.179,E2 -401.179} C_VEL
LIN {X 0,Y 608.473,Z 355.314,A -85,B 0,C 180,E1 -403.869,E2 -403.869} C_VEL
LIN {X 0,Y 608.442,Z 355.317,A -85,B 0,C 180,E1 -406.694,E2 -406.694} C_VEL
LIN {X 0,Y 608.411,Z 355.319,A -85,B 0,C 180,E1 -408.819,E2 -408.819} C_VEL
LIN {X 0,Y 608.463,Z 355.317,A -85,B 0,C 180,E1 -411.76,E2 -411.76} C_VEL
LIN {X 0,Y 608.403,Z 355.32,A -85,B 0,C 180,E1 -414.719,E2 -414.719} C_VEL
LIN {X 0,Y 608.438,Z 355.319,A -85,B 0,C 180,E1 -417.481,E2 -417.481} C_VEL
LIN {X 0,Y 608.433,Z 355.32,A -85,B 0,C 180,E1 -420.218,E2 -420.218} C_VEL
LIN {X 0,Y 608.478,Z 355.497,A -85,B 0,C 180,E1 -421.649,E2 -421.649} C_VEL
LIN {X 0,Y 608.905,Z 358.269,A -85,B 0,C 180,E1 -421.943,E2 -421.943} C_VEL
LIN {X 0,Y 608.802,Z 390.533,A -85,B 0,C 180,E1 -424.714,E2 -424.714} C_VEL
LIN {X 0,Y 608.718,Z 423.286,A -85,B 0,C 180,E1 -427.465,E2 -427.465} C_VEL
LIN {X 0,Y 608.633,Z 455.063,A -85,B 0,C 180,E1 -430.083,E2 -430.083} C_VEL
LIN {X 0,Y 608.634,Z 472.757,A -85,B 0,C 180,E1 -431.507,E2 -431.507} C_VEL
LIN {X 0,Y 608.759,Z 507.298,A -85,B 0,C 180,E1 -431.946,E2 -431.946} C_VEL
LIN {X 0,Y 608.693,Z 640.913,A -85,B 0,C 180,E1 -433.578,E2 -433.578} C_VEL
LIN {X 0,Y 608.651,Z 656.682,A -85,B 0,C 180,E1 -433.911,E2 -433.911} C_VEL
LIN {X 0,Y 608.619,Z 672.027,A -85,B 0,C 180,E1 -434.382,E2 -434.382} C_VEL
LIN {X 0,Y 608.605,Z 685.736,A -85,B 0,C 180,E1 -434.94,E2 -434.94} C_VEL
LIN {X 0,Y 608.573,Z 699.22,A -85,B 0,C 180,E1 -435.623,E2 -435.623} C_VEL
LIN {X 0,Y 608.554,Z 711.652,A -85,B 0,C 180,E1 -436.39,E2 -436.39} C_VEL
LIN {X 0,Y 608.528,Z 724.272,A -85,B 0,C 180,E1 -437.323,E2 -437.323} C_VEL
LIN {X 0,Y 608.496,Z 735.738,A -85,B 0,C 180,E1 -438.338,E2 -438.338} C_VEL
LIN {X 0,Y 608.475,Z 745.38,A -85,B 0,C 180,E1 -439.349,E2 -439.349} C_VEL
LIN {X 0,Y 608.477,Z 754.847,A -85,B 0,C 180,E1 -440.526,E2 -440.526} C_VEL
LIN {X 0,Y 608.456,Z 762.723,A -85,B 0,C 180,E1 -441.698,E2 -441.698} C_VEL
LIN {X 0,Y 608.442,Z 770.083,A -85,B 0,C 180,E1 -443.033,E2 -443.033} C_VEL
LIN {X 0,Y 608.449,Z 775.92,A -85,B 0,C 180,E1 -444.365,E2 -444.365} C_VEL
LIN {X 0,Y 608.427,Z 779.38,A -85,B 0,C 180,E1 -445.361,E2 -445.361} C_VEL
LIN {X 0,Y 608.421,Z 782.883,A -85,B 0,C 180,E1 -446.688,E2 -446.688} C_VEL
LIN {X 0,Y 608.441,Z 785.19,A -85,B 0,C 180,E1 -448.013,E2 -448.013} C_VEL
LIN {X 0,Y 608.436,Z 786.35,A -85,B 0,C 180,E1 -449.337,E2 -449.337} C_VEL
LIN {X 0,Y 608.436,Z 786.351,A -85,B 0,C 180,E1 -450.661,E2 -450.661} C_VEL
LIN {X 0,Y 608.44,Z 785.192,A -85,B 0,C 180,E1 -451.985,E2 -451.985} C_VEL
LIN {X 0,Y 608.421,Z 782.888,A -85,B 0,C 180,E1 -453.31,E2 -453.31} C_VEL
LIN {X 0,Y 608.427,Z 779.386,A -85,B 0,C 180,E1 -454.637,E2 -454.637} C_VEL
LIN {X 0,Y 608.431,Z 774.612,A -85,B 0,C 180,E1 -455.966,E2 -455.966} C_VEL
LIN {X 0,Y 608.458,Z 768.432,A -85,B 0,C 180,E1 -457.298,E2 -457.298} C_VEL
LIN {X 0,Y 608.465,Z 760.662,A -85,B 0,C 180,E1 -458.635,E2 -458.635} C_VEL
LIN {X 0,Y 608.471,Z 752.379,A -85,B 0,C 180,E1 -459.808,E2 -459.808} C_VEL
LIN {X 0,Y 608.491,Z 741.657,A -85,B 0,C 180,E1 -461.062,E2 -461.062} C_VEL
LIN {X 0,Y 608.522,Z 730.288,A -85,B 0,C 180,E1 -462.167,E2 -462.167} C_VEL
LIN {X 0,Y 608.547,Z 718.87,A -85,B 0,C 180,E1 -463.098,E2 -463.098} C_VEL
LIN {X 0,Y 608.56,Z 706.466,A -85,B 0,C 180,E1 -463.949,E2 -463.949} C_VEL
LIN {X 0,Y 608.587,Z 692.885,A -85,B 0,C 180,E1 -464.716,E2 -464.716} C_VEL
LIN {X 0,Y 608.631,Z 678.824,A -85,B 0,C 180,E1 -465.358,E2 -465.358} C_VEL
LIN {X 0,Y 608.634,Z 664.34,A -85,B 0,C 180,E1 -465.873,E2 -465.873} C_VEL
LIN {X 0,Y 608.675,Z 648.975,A -85,B 0,C 180,E1 -466.271,E2 -466.271} C_VEL
LIN {X 0,Y 608.7,Z 633.339,A -85,B 0,C 180,E1 -466.53,E2 -466.53} C_VEL
LIN {X 0,Y 608.754,Z 473.653,A -85,B 0,C 180,E1 -468.468,E2 -468.468} C_VEL
LIN {X 0,Y 608.605,Z 471.851,A -85,B 0,C 180,E1 -468.553,E2 -468.553} C_VEL
LIN {X 0,Y 608.7,Z 436.806,A -85,B 0,C 180,E1 -471.415,E2 -471.415} C_VEL
LIN {X 0,Y 608.769,Z 403.22,A -85,B 0,C 180,E1 -474.214,E2 -474.214} C_VEL
LIN {X 0,Y 608.872,Z 369.803,A -85,B 0,C 180,E1 -477.059,E2 -477.059} C_VEL
LIN {X 0,Y 608.878,Z 357.22,A -85,B 0,C 180,E1 -478.15,E2 -478.15} C_VEL
LIN {X 0,Y 608.457,Z 355.431,A -85,B 0,C 180,E1 -478.372,E2 -478.372} C_VEL
LIN {X 0,Y 608.445,Z 355.319,A -85,B 0,C 180,E1 -480.545,E2 -480.545} C_VEL
LIN {X 0,Y 608.416,Z 355.319,A -85,B 0,C 180,E1 -482.88,E2 -482.88} C_VEL
LIN {X 0,Y 608.392,Z 355.32,A -85,B 0,C 180,E1 -485.279,E2 -485.279} C_VEL
LIN {X 0,Y 608.451,Z 355.323,A -85,B 0,C 180,E1 -488.238,E2 -488.238} C_VEL
LIN {X 0,Y 608.433,Z 355.326,A -85,B 0,C 180,E1 -490.327,E2 -490.327} C_VEL
LIN {X 0,Y 608.394,Z 355.321,A -85,B 0,C 180,E1 -492.963,E2 -492.963} C_VEL
LIN {X 0,Y 608.395,Z 355.319,A -85,B 0,C 180,E1 -495.199,E2 -495.199} C_VEL
LIN {X 0,Y 608.426,Z 355.319,A -85,B 0,C 180,E1 -497.936,E2 -497.936} C_VEL
LIN {X 0,Y 608.412,Z 355.322,A -85,B 0,C 180,E1 -500.707,E2 -500.707} C_VEL
LIN {X 0,Y 608.391,Z 355.32,A -85,B 0,C 180,E1 -503.081,E2 -503.081} C_VEL
LIN {X 0,Y 608.411,Z 355.317,A -85,B 0,C 180,E1 -505.527,E2 -505.527} C_VEL
LIN {X 0,Y 608.426,Z 355.318,A -85,B 0,C 180,E1 -507.903,E2 -507.903} C_VEL
LIN {X 0,Y 608.46,Z 355.319,A -85,B 0,C 180,E1 -510.22,E2 -510.22} C_VEL
LIN {X 0,Y 608.386,Z 355.321,A -85,B 0,C 180,E1 -513.223,E2 -513.223} C_VEL
LIN {X 0,Y 608.399,Z 355.318,A -85,B 0,C 180,E1 -515.427,E2 -515.427} C_VEL
LIN {X 0,Y 608.445,Z 355.321,A -85,B 0,C 180,E1 -518.308,E2 -518.308} C_VEL
LIN {X 0,Y 608.398,Z 355.319,A -85,B 0,C 180,E1 -521.299,E2 -521.299} C_VEL
LIN {X 0,Y 608.414,Z 355.319,A -85,B 0,C 180,E1 -523.905,E2 -523.905} C_VEL
LIN {X 0,Y 608.432,Z 355.323,A -85,B 0,C 180,E1 -526.643,E2 -526.643} C_VEL
LIN {X 0,Y 608.397,Z 355.319,A -85,B 0,C 180,E1 -529.349,E2 -529.349} C_VEL
LIN {X 0,Y 608.392,Z 355.319,A -85,B 0,C 180,E1 -531.363,E2 -531.363} C_VEL
LIN {X 0,Y 608.418,Z 355.319,A -85,B 0,C 180,E1 -534.033,E2 -534.033} C_VEL
LIN {X 0,Y 608.459,Z 355.32,A -85,B 0,C 180,E1 -536.689,E2 -536.689} C_VEL
LIN {X 0,Y 608.395,Z 355.32,A -85,B 0,C 180,E1 -539.338,E2 -539.338} C_VEL
LIN {X 0,Y 608.406,Z 355.318,A -85,B 0,C 180,E1 -541.324,E2 -541.324} C_VEL
LIN {X 0,Y 608.386,Z 355.321,A -85,B 0,C 180,E1 -543.311,E2 -543.311} C_VEL
LIN {X 0,Y 608.403,Z 355.319,A -85,B 0,C 180,E1 -545.302,E2 -545.302} C_VEL
LIN {X 0,Y 608.398,Z 355.32,A -85,B 0,C 180,E1 -547.3,E2 -547.3} C_VEL
LIN {X 0,Y 608.402,Z 355.318,A -85,B 0,C 180,E1 -549.47,E2 -549.47} C_VEL
LIN {X 0,Y 607.726,Z 355.405,A -85,B 0,C 180,E1 -550.022,E2 -550.022} C_VEL
LIN {X 0,Y 604.875,Z 355.763,A -85,B 0,C 180,E1 -550.92,E2 -550.92} C_VEL
LIN {X 0,Y 602.478,Z 356.059,A -85,B 0,C 180,E1 -551.641,E2 -551.641} C_VEL
LIN {X 0,Y 601.456,Z 356.186,A -85,B 0,C 180,E1 -552.198,E2 -552.198} C_VEL
LIN {X 0,Y 601.376,Z 356.196,A -85,B 0,C 180,E1 -552.386,E2 -552.386} C_VEL
LIN {X 0,Y 601.401,Z 356.197,A -85,B 0,C 180,E1 -554.898,E2 -554.898} C_VEL
LIN {X 0,Y 601.406,Z 356.195,A -85,B 0,C 180,E1 -556.987,E2 -556.987} C_VEL
LIN {X 0,Y 601.359,Z 356.196,A -85,B 0,C 180,E1 -559.811,E2 -559.811} C_VEL
LIN {X 0,Y 601.366,Z 356.195,A -85,B 0,C 180,E1 -561.961,E2 -561.961} C_VEL
LIN {X 0,Y 601.363,Z 356.202,A -85,B 0,C 180,E1 -564.88,E2 -564.88} C_VEL
LIN {X 0,Y 601.362,Z 356.197,A -85,B 0,C 180,E1 -567.356,E2 -567.356} C_VEL
LIN {X 0,Y 601.359,Z 356.197,A -85,B 0,C 180,E1 -569.396,E2 -569.396} C_VEL
LIN {X 0,Y 601.368,Z 356.195,A -85,B 0,C 180,E1 -571.729,E2 -571.729} C_VEL
LIN {X 0,Y 601.397,Z 356.193,A -85,B 0,C 180,E1 -574.121,E2 -574.121} C_VEL
LIN {X 0,Y 601.38,Z 356.201,A -85,B 0,C 180,E1 -576.585,E2 -576.585} C_VEL
LIN {X 0,Y 601.373,Z 356.195,A -85,B 0,C 180,E1 -579.53,E2 -579.53} C_VEL
LIN {X 0,Y 601.364,Z 356.194,A -85,B 0,C 180,E1 -581.77,E2 -581.77} C_VEL
LIN {X 0,Y 601.386,Z 356.198,A -85,B 0,C 180,E1 -584.534,E2 -584.534} C_VEL
LIN {X 0,Y 601.356,Z 356.199,A -85,B 0,C 180,E1 -587.327,E2 -587.327} C_VEL
LIN {X 0,Y 601.365,Z 356.195,A -85,B 0,C 180,E1 -590.003,E2 -590.003} C_VEL
LIN {X 0,Y 601.424,Z 356.195,A -85,B 0,C 180,E1 -592.62,E2 -592.62} C_VEL
LIN {X 0,Y 601.387,Z 356.191,A -85,B 0,C 180,E1 -595.881,E2 -595.881} C_VEL
LIN {X 0,Y 601.383,Z 356.199,A -85,B 0,C 180,E1 -598.551,E2 -598.551} C_VEL
LIN {X 0,Y 601.434,Z 356.382,A -85,B 0,C 180,E1 -600.489,E2 -600.489} C_VEL
LIN {X 0,Y 602.146,Z 358.848,A -85,B 0,C 180,E1 -600.791,E2 -600.791} C_VEL
LIN {X 0,Y 602.157,Z 378.26,A -85,B 0,C 180,E1 -602.652,E2 -602.652} C_VEL
LIN {X 0,Y 602.012,Z 406.512,A -85,B 0,C 180,E1 -605.298,E2 -605.298} C_VEL
LIN {X 0,Y 601.905,Z 434.67,A -85,B 0,C 180,E1 -607.883,E2 -607.883} C_VEL
LIN {X 0,Y 601.745,Z 466.349,A -85,B 0,C 180,E1 -610.736,E2 -610.736} C_VEL
LIN {X 0,Y 601.761,Z 473.318,A -85,B 0,C 180,E1 -611.338,E2 -611.338} C_VEL
LIN {X 0,Y 602.036,Z 477.702,A -85,B 0,C 180,E1 -611.417,E2 -611.417} C_VEL
LIN {X 0,Y 601.886,Z 641.491,A -85,B 0,C 180,E1 -613.442,E2 -613.442} C_VEL
LIN {X 0,Y 601.829,Z 657.509,A -85,B 0,C 180,E1 -613.791,E2 -613.791} C_VEL
LIN {X 0,Y 601.79,Z 672.034,A -85,B 0,C 180,E1 -614.246,E2 -614.246} C_VEL
LIN {X 0,Y 601.705,Z 686.705,A -85,B 0,C 180,E1 -614.852,E2 -614.852} C_VEL
LIN {X 0,Y 601.657,Z 700.003,A -85,B 0,C 180,E1 -615.543,E2 -615.543} C_VEL
LIN {X 0,Y 601.604,Z 712.817,A -85,B 0,C 180,E1 -616.353,E2 -616.353} C_VEL
LIN {X 0,Y 601.541,Z 724.806,A -85,B 0,C 180,E1 -617.261,E2 -617.261} C_VEL
LIN {X 0,Y 601.488,Z 735.297,A -85,B 0,C 180,E1 -618.202,E2 -618.202} C_VEL
LIN {X 0,Y 601.43,Z 745.01,A -85,B 0,C 180,E1 -619.225,E2 -619.225} C_VEL
LIN {X 0,Y 601.428,Z 754.538,A -85,B 0,C 180,E1 -620.416,E2 -620.416} C_VEL
LIN {X 0,Y 601.378,Z 762.47,A -85,B 0,C 180,E1 -621.601,E2 -621.601} C_VEL
LIN {X 0,Y 601.367,Z 769.879,A -85,B 0,C 180,E1 -622.953,E2 -622.953} C_VEL
LIN {X 0,Y 601.371,Z 775.764,A -85,B 0,C 180,E1 -624.3,E2 -624.3} C_VEL
LIN {X 0,Y 601.328,Z 779.245,A -85,B 0,C 180,E1 -625.308,E2 -625.308} C_VEL
LIN {X 0,Y 601.336,Z 782.791,A -85,B 0,C 180,E1 -626.651,E2 -626.651} C_VEL
LIN {X 0,Y 601.342,Z 785.14,A -85,B 0,C 180,E1 -627.992,E2 -627.992} C_VEL
LIN {X 0,Y 601.334,Z 786.337,A -85,B 0,C 180,E1 -629.331,E2 -629.331} C_VEL
LIN {X 0,Y 601.335,Z 786.361,A -85,B 0,C 180,E1 -630.671,E2 -630.671} C_VEL
LIN {X 0,Y 601.343,Z 785.243,A -85,B 0,C 180,E1 -632.01,E2 -632.01} C_VEL
LIN {X 0,Y 601.339,Z 782.98,A -85,B 0,C 180,E1 -633.351,E2 -633.351} C_VEL
LIN {X 0,Y 601.328,Z 779.522,A -85,B 0,C 180,E1 -634.694,E2 -634.694} C_VEL
LIN {X 0,Y 601.356,Z 774.795,A -85,B 0,C 180,E1 -636.039,E2 -636.039} C_VEL
LIN {X 0,Y 601.366,Z 768.659,A -85,B 0,C 180,E1 -637.387,E2 -637.387} C_VEL
LIN {X 0,Y 601.388,Z 760.942,A -85,B 0,C 180,E1 -638.739,E2 -638.739} C_VEL
LIN {X 0,Y 601.428,Z 752.702,A -85,B 0,C 180,E1 -639.926,E2 -639.926} C_VEL
LIN {X 0,Y 601.444,Z 742.354,A -85,B 0,C 180,E1 -641.165,E2 -641.165} C_VEL
LIN {X 0,Y 601.503,Z 730.777,A -85,B 0,C 180,E1 -642.313,E2 -642.313} C_VEL
LIN {X 0,Y 601.56,Z 718.291,A -85,B 0,C 180,E1 -643.341,E2 -643.341} C_VEL
LIN {X 0,Y 601.644,Z 705.762,A -85,B 0,C 180,E1 -644.201,E2 -644.201} C_VEL
LIN {X 0,Y 601.685,Z 692.01,A -85,B 0,C 180,E1 -644.978,E2 -644.978} C_VEL
LIN {X 0,Y 601.754,Z 677.701,A -85,B 0,C 180,E1 -645.627,E2 -645.627} C_VEL
LIN {X 0,Y 601.798,Z 662.847,A -85,B 0,C 180,E1 -646.147,E2 -646.147} C_VEL
LIN {X 0,Y 601.862,Z 647.077,A -85,B 0,C 180,E1 -646.543,E2 -646.543} C_VEL
LIN {X 0,Y 601.909,Z 630.578,A -85,B 0,C 180,E1 -646.801,E2 -646.801} C_VEL
LIN {X 0,Y 601.933,Z 474.713,A -85,B 0,C 180,E1 -648.714,E2 -648.714} C_VEL
LIN {X 0,Y 601.751,Z 473.184,A -85,B 0,C 180,E1 -648.76,E2 -648.76} C_VEL
LIN {X 0,Y 601.837,Z 443.537,A -85,B 0,C 180,E1 -651.404,E2 -651.404} C_VEL
LIN {X 0,Y 602.013,Z 412.178,A -85,B 0,C 180,E1 -654.267,E2 -654.267} C_VEL
LIN {X 0,Y 602.13,Z 384.047,A -85,B 0,C 180,E1 -656.891,E2 -656.891} C_VEL
LIN {X 0,Y 602.281,Z 360.429,A -85,B 0,C 180,E1 -659.139,E2 -659.139} C_VEL
LIN {X 0,Y 601.424,Z 356.457,A -85,B 0,C 180,E1 -659.586,E2 -659.586} C_VEL
LIN {X 0,Y 601.345,Z 356.203,A -85,B 0,C 180,E1 -660.169,E2 -660.169} C_VEL
LIN {X 0,Y 601.379,Z 356.198,A -85,B 0,C 180,E1 -662.709,E2 -662.709} C_VEL
LIN {X 0,Y 601.341,Z 356.201,A -85,B 0,C 180,E1 -665.759,E2 -665.759} C_VEL
LIN {X 0,Y 601.337,Z 356.199,A -85,B 0,C 180,E1 -668.275,E2 -668.275} C_VEL
LIN {X 0,Y 601.371,Z 356.2,A -85,B 0,C 180,E1 -670.879,E2 -670.879} C_VEL
LIN {X 0,Y 601.407,Z 356.194,A -85,B 0,C 180,E1 -673.589,E2 -673.589} C_VEL
LIN {X 0,Y 601.378,Z 356.194,A -85,B 0,C 180,E1 -676.433,E2 -676.433} C_VEL
LIN {X 0,Y 601.401,Z 356.196,A -85,B 0,C 180,E1 -679.429,E2 -679.429} C_VEL
LIN {X 0,Y 601.354,Z 356.199,A -85,B 0,C 180,E1 -681.727,E2 -681.727} C_VEL
LIN {X 0,Y 601.357,Z 356.196,A -85,B 0,C 180,E1 -684.243,E2 -684.243} C_VEL
LIN {X 0,Y 601.372,Z 356.197,A -85,B 0,C 180,E1 -686.683,E2 -686.683} C_VEL
LIN {X 0,Y 601.396,Z 356.201,A -85,B 0,C 180,E1 -689.057,E2 -689.057} C_VEL
LIN {X 0,Y 601.424,Z 356.195,A -85,B 0,C 180,E1 -691.373,E2 -691.373} C_VEL
LIN {X 0,Y 601.37,Z 356.195,A -85,B 0,C 180,E1 -694.142,E2 -694.142} C_VEL
LIN {X 0,Y 601.37,Z 356.197,A -85,B 0,C 180,E1 -696.588,E2 -696.588} C_VEL
LIN {X 0,Y 601.423,Z 356.194,A -85,B 0,C 180,E1 -699.478,E2 -699.478} C_VEL
LIN {X 0,Y 601.443,Z 356.342,A -85,B 0,C 180,E1 -701.033,E2 -701.033} C_VEL
LIN {X 0,Y 601.492,Z 368.559,A -85,B 0,C 180,E1 -703.016,E2 -703.016} C_VEL
LIN {X 0,Y 601.483,Z 375.277,A -85,B 0,C 180,E1 -704.063,E2 -704.063} C_VEL
LIN {X 0,Y 601.807,Z 377.483,A -85,B 0,C 180,E1 -704.137,E2 -704.137} C_VEL
LIN {X 0,Y 601.749,Z 511.427,A -85,B 0,C 180,E1 -705.774,E2 -705.774} C_VEL
LIN {X 0,Y 601.722,Z 525.539,A -85,B 0,C 180,E1 -706.081,E2 -706.081} C_VEL
LIN {X 0,Y 601.669,Z 539.675,A -85,B 0,C 180,E1 -706.533,E2 -706.533} C_VEL
LIN {X 0,Y 601.603,Z 552.728,A -85,B 0,C 180,E1 -707.09,E2 -707.09} C_VEL
LIN {X 0,Y 601.546,Z 565.358,A -85,B 0,C 180,E1 -707.775,E2 -707.775} C_VEL
LIN {X 0,Y 601.505,Z 576.862,A -85,B 0,C 180,E1 -708.543,E2 -708.543} C_VEL
LIN {X 0,Y 601.482,Z 587.42,A -85,B 0,C 180,E1 -709.395,E2 -709.395} C_VEL
LIN {X 0,Y 601.431,Z 597.903,A -85,B 0,C 180,E1 -710.415,E2 -710.415} C_VEL
LIN {X 0,Y 601.406,Z 606.556,A -85,B 0,C 180,E1 -711.431,E2 -711.431} C_VEL
LIN {X 0,Y 601.392,Z 614.838,A -85,B 0,C 180,E1 -712.614,E2 -712.614} C_VEL
LIN {X 0,Y 601.361,Z 620.523,A -85,B 0,C 180,E1 -713.606,E2 -713.606} C_VEL
LIN {X 0,Y 601.355,Z 625.382,A -85,B 0,C 180,E1 -714.635,E2 -714.635} C_VEL
LIN {X 0,Y 601.344,Z 630.304,A -85,B 0,C 180,E1 -715.979,E2 -715.979} C_VEL
LIN {X 0,Y 601.324,Z 633.737,A -85,B 0,C 180,E1 -717.32,E2 -717.32} C_VEL
LIN {X 0,Y 601.346,Z 635.779,A -85,B 0,C 180,E1 -718.661,E2 -718.661} C_VEL
LIN {X 0,Y 601.332,Z 636.495,A -85,B 0,C 180,E1 -720,E2 -720} C_VEL
LIN {X 0,Y 601.342,Z 635.882,A -85,B 0,C 180,E1 -721.339,E2 -721.339} C_VEL
LIN {X 0,Y 601.324,Z 633.928,A -85,B 0,C 180,E1 -722.679,E2 -722.679} C_VEL
LIN {X 0,Y 601.345,Z 630.586,A -85,B 0,C 180,E1 -724.021,E2 -724.021} C_VEL
LIN {X 0,Y 601.354,Z 625.762,A -85,B 0,C 180,E1 -725.365,E2 -725.365} C_VEL
LIN {X 0,Y 601.374,Z 619.871,A -85,B 0,C 180,E1 -726.605,E2 -726.605} C_VEL
LIN {X 0,Y 601.386,Z 613.223,A -85,B 0,C 180,E1 -727.723,E2 -727.723} C_VEL
LIN {X 0,Y 601.411,Z 604.565,A -85,B 0,C 180,E1 -728.907,E2 -728.907} C_VEL
LIN {X 0,Y 601.431,Z 595.521,A -85,B 0,C 180,E1 -729.925,E2 -729.925} C_VEL
LIN {X 0,Y 601.497,Z 585.362,A -85,B 0,C 180,E1 -730.876,E2 -730.876} C_VEL
LIN {X 0,Y 601.547,Z 573.384,A -85,B 0,C 180,E1 -731.798,E2 -731.798} C_VEL
LIN {X 0,Y 601.588,Z 561.042,A -85,B 0,C 180,E1 -732.567,E2 -732.567} C_VEL
LIN {X 0,Y 601.631,Z 549.17,A -85,B 0,C 180,E1 -733.167,E2 -733.167} C_VEL
LIN {X 0,Y 601.687,Z 535.229,A -85,B 0,C 180,E1 -733.714,E2 -733.714} C_VEL
LIN {X 0,Y 601.702,Z 521.331,A -85,B 0,C 180,E1 -734.113,E2 -734.113} C_VEL
LIN {X 0,Y 601.75,Z 507.371,A -85,B 0,C 180,E1 -734.376,E2 -734.376} C_VEL
LIN {X 0,Y 601.719,Z 376.756,A -85,B 0,C 180,E1 -735.966,E2 -735.966} C_VEL
LIN {X 0,Y 601.489,Z 375.085,A -85,B 0,C 180,E1 -736.046,E2 -736.046} C_VEL
LIN {X 0,Y 601.531,Z 357.483,A -85,B 0,C 180,E1 -738.849,E2 -738.849} C_VEL
LIN {X 0,Y 601.43,Z 356.263,A -85,B 0,C 180,E1 -739.098,E2 -739.098} C_VEL
LIN {X 0,Y 601.407,Z 356.196,A -85,B 0,C 180,E1 -741.239,E2 -741.239} C_VEL
LIN {X 0,Y 601.446,Z 356.187,A -85,B 0,C 180,E1 -744.141,E2 -744.141} C_VEL
LIN {X 0,Y 601.448,Z 356.19,A -85,B 0,C 180,E1 -747.111,E2 -747.111} C_VEL
LIN {X 0,Y 601.422,Z 356.19,A -85,B 0,C 180,E1 -749.393,E2 -749.393} C_VEL
LIN {X 0,Y 601.403,Z 356.191,A -85,B 0,C 180,E1 -751.727,E2 -751.727} C_VEL
LIN {X 0,Y 601.431,Z 356.191,A -85,B 0,C 180,E1 -754.118,E2 -754.118} C_VEL
LIN {X 0,Y 601.396,Z 356.2,A -85,B 0,C 180,E1 -756.583,E2 -756.583} C_VEL
LIN {X 0,Y 601.399,Z 356.192,A -85,B 0,C 180,E1 -759.127,E2 -759.127} C_VEL
LIN {X 0,Y 601.423,Z 356.191,A -85,B 0,C 180,E1 -761.765,E2 -761.765} C_VEL
LIN {X 0,Y 601.401,Z 356.197,A -85,B 0,C 180,E1 -764.532,E2 -764.532} C_VEL
LIN {X 0,Y 601.386,Z 356.194,A -85,B 0,C 180,E1 -767.412,E2 -767.412} C_VEL
LIN {X 0,Y 601.398,Z 356.201,A -85,B 0,C 180,E1 -770.003,E2 -770.003} C_VEL
LIN {X 0,Y 601.391,Z 356.194,A -85,B 0,C 180,E1 -772.623,E2 -772.623} C_VEL
LIN {X 0,Y 601.363,Z 356.197,A -85,B 0,C 180,E1 -775.064,E2 -775.064} C_VEL
LIN {X 0,Y 601.407,Z 356.195,A -85,B 0,C 180,E1 -777.482,E2 -777.482} C_VEL
LIN {X 0,Y 601.405,Z 356.201,A -85,B 0,C 180,E1 -779.855,E2 -779.855} C_VEL
LIN {X 0,Y 601.411,Z 356.409,A -85,B 0,C 180,E1 -781.371,E2 -781.371} C_VEL
LIN {X 0,Y 602.259,Z 359.344,A -85,B 0,C 180,E1 -781.7,E2 -781.7} C_VEL
LIN {X 0,Y 602.12,Z 387.503,A -85,B 0,C 180,E1 -784.152,E2 -784.152} C_VEL
LIN {X 0,Y 601.974,Z 419.575,A -85,B 0,C 180,E1 -786.885,E2 -786.885} C_VEL
LIN {X 0,Y 601.834,Z 450.761,A -85,B 0,C 180,E1 -789.492,E2 -789.492} C_VEL
LIN {X 0,Y 601.79,Z 472.904,A -85,B 0,C 180,E1 -791.295,E2 -791.295} C_VEL
LIN {X 0,Y 602.033,Z 478.92,A -85,B 0,C 180,E1 -791.387,E2 -791.387} C_VEL
LIN {X 0,Y 601.893,Z 641.21,A -85,B 0,C 180,E1 -793.392,E2 -793.392} C_VEL
LIN {X 0,Y 601.829,Z 656.682,A -85,B 0,C 180,E1 -793.723,E2 -793.723} C_VEL
LIN {X 0,Y 601.768,Z 672.027,A -85,B 0,C 180,E1 -794.2,E2 -794.2} C_VEL
LIN {X 0,Y 601.721,Z 685.738,A -85,B 0,C 180,E1 -794.763,E2 -794.763} C_VEL
LIN {X 0,Y 601.659,Z 699.216,A -85,B 0,C 180,E1 -795.454,E2 -795.454} C_VEL
LIN {X 0,Y 601.617,Z 712.443,A -85,B 0,C 180,E1 -796.283,E2 -796.283} C_VEL
LIN {X 0,Y 601.531,Z 724.274,A -85,B 0,C 180,E1 -797.173,E2 -797.173} C_VEL
LIN {X 0,Y 601.488,Z 735.739,A -85,B 0,C 180,E1 -798.2,E2 -798.2} C_VEL
LIN {X 0,Y 601.43,Z 745.381,A -85,B 0,C 180,E1 -799.223,E2 -799.223} C_VEL
LIN {X 0,Y 601.428,Z 754.847,A -85,B 0,C 180,E1 -800.414,E2 -800.414} C_VEL
LIN {X 0,Y 601.368,Z 762.724,A -85,B 0,C 180,E1 -801.599,E2 -801.599} C_VEL
LIN {X 0,Y 601.369,Z 770.083,A -85,B 0,C 180,E1 -802.951,E2 -802.951} C_VEL
LIN {X 0,Y 601.371,Z 775.921,A -85,B 0,C 180,E1 -804.298,E2 -804.298} C_VEL
LIN {X 0,Y 601.33,Z 779.38,A -85,B 0,C 180,E1 -805.306,E2 -805.306} C_VEL
LIN {X 0,Y 601.337,Z 782.884,A -85,B 0,C 180,E1 -806.649,E2 -806.649} C_VEL
LIN {X 0,Y 601.339,Z 785.19,A -85,B 0,C 180,E1 -807.99,E2 -807.99} C_VEL
LIN {X 0,Y 601.337,Z 786.35,A -85,B 0,C 180,E1 -809.329,E2 -809.329} C_VEL
LIN {X 0,Y 601.337,Z 786.351,A -85,B 0,C 180,E1 -810.669,E2 -810.669} C_VEL
LIN {X 0,Y 601.339,Z 785.193,A -85,B 0,C 180,E1 -812.008,E2 -812.008} C_VEL
LIN {X 0,Y 601.337,Z 782.888,A -85,B 0,C 180,E1 -813.349,E2 -813.349} C_VEL
LIN {X 0,Y 601.33,Z 779.387,A -85,B 0,C 180,E1 -814.692,E2 -814.692} C_VEL
LIN {X 0,Y 601.352,Z 774.612,A -85,B 0,C 180,E1 -816.037,E2 -816.037} C_VEL
LIN {X 0,Y 601.381,Z 768.432,A -85,B 0,C 180,E1 -817.385,E2 -817.385} C_VEL
LIN {X 0,Y 601.387,Z 760.661,A -85,B 0,C 180,E1 -818.737,E2 -818.737} C_VEL
LIN {X 0,Y 601.427,Z 752.379,A -85,B 0,C 180,E1 -819.924,E2 -819.924} C_VEL
LIN {X 0,Y 601.459,Z 741.939,A -85,B 0,C 180,E1 -821.164,E2 -821.164} C_VEL
LIN {X 0,Y 601.513,Z 732.205,A -85,B 0,C 180,E1 -822.139,E2 -822.139} C_VEL
LIN {X 0,Y 601.57,Z 720.03,A -85,B 0,C 180,E1 -823.167,E2 -823.167} C_VEL
LIN {X 0,Y 601.603,Z 708.095,A -85,B 0,C 180,E1 -824.01,E2 -824.01} C_VEL
LIN {X 0,Y 601.661,Z 694.551,A -85,B 0,C 180,E1 -824.803,E2 -824.803} C_VEL
LIN {X 0,Y 601.762,Z 679.872,A -85,B 0,C 180,E1 -825.494,E2 -825.494} C_VEL
LIN {X 0,Y 601.785,Z 665.654,A -85,B 0,C 180,E1 -826.015,E2 -826.015} C_VEL
LIN {X 0,Y 601.863,Z 650.621,A -85,B 0,C 180,E1 -826.421,E2 -826.421} C_VEL
LIN {X 0,Y 601.898,Z 635.559,A -85,B 0,C 180,E1 -826.691,E2 -826.691} C_VEL
LIN {X 0,Y 602.014,Z 474.406,A -85,B 0,C 180,E1 -828.669,E2 -828.669} C_VEL
LIN {X 0,Y 601.776,Z 472.612,A -85,B 0,C 180,E1 -828.719,E2 -828.719} C_VEL
LIN {X 0,Y 601.901,Z 437.882,A -85,B 0,C 180,E1 -831.579,E2 -831.579} C_VEL
LIN {X 0,Y 602.05,Z 404.155,A -85,B 0,C 180,E1 -834.422,E2 -834.422} C_VEL
LIN {X 0,Y 602.249,Z 370.156,A -85,B 0,C 180,E1 -837.35,E2 -837.35} C_VEL
LIN {X 0,Y 602.257,Z 359.371,A -85,B 0,C 180,E1 -838.297,E2 -838.297} C_VEL
LIN {X 0,Y 601.394,Z 356.338,A -85,B 0,C 180,E1 -838.648,E2 -838.648} C_VEL
LIN {X 0,Y 601.377,Z 356.195,A -85,B 0,C 180,E1 -840.943,E2 -840.943} C_VEL
LIN {X 0,Y 601.366,Z 356.196,A -85,B 0,C 180,E1 -843.316,E2 -843.316} C_VEL
LIN {X 0,Y 601.378,Z 356.204,A -85,B 0,C 180,E1 -846.258,E2 -846.258} C_VEL
LIN {X 0,Y 601.363,Z 356.196,A -85,B 0,C 180,E1 -849.128,E2 -849.128} C_VEL
LIN {X 0,Y 601.399,Z 356.193,A -85,B 0,C 180,E1 -851.765,E2 -851.765} C_VEL
LIN {X 0,Y 601.386,Z 356.2,A -85,B 0,C 180,E1 -854.531,E2 -854.531} C_VEL
LIN {X 0,Y 601.337,Z 356.197,A -85,B 0,C 180,E1 -857.323,E2 -857.323} C_VEL
LIN {X 0,Y 601.384,Z 356.192,A -85,B 0,C 180,E1 -859.428,E2 -859.428} C_VEL
LIN {X 0,Y 601.354,Z 356.198,A -85,B 0,C 180,E1 -861.727,E2 -861.727} C_VEL
LIN {X 0,Y 601.369,Z 356.202,A -85,B 0,C 180,E1 -864.244,E2 -864.244} C_VEL
LIN {X 0,Y 601.401,Z 356.196,A -85,B 0,C 180,E1 -866.685,E2 -866.685} C_VEL
LIN {X 0,Y 601.371,Z 356.195,A -85,B 0,C 180,E1 -869.055,E2 -869.055} C_VEL
LIN {X 0,Y 601.371,Z 356.194,A -85,B 0,C 180,E1 -871.37,E2 -871.37} C_VEL
LIN {X 0,Y 601.428,Z 356.197,A -85,B 0,C 180,E1 -874.382,E2 -874.382} C_VEL
LIN {X 0,Y 601.385,Z 356.192,A -85,B 0,C 180,E1 -877.397,E2 -877.397} C_VEL
LIN {X 0,Y 601.371,Z 356.2,A -85,B 0,C 180,E1 -880.189,E2 -880.189} C_VEL
LIN {X 0,Y 601.359,Z 356.198,A -85,B 0,C 180,E1 -883.012,E2 -883.012} C_VEL
LIN {X 0,Y 601.384,Z 356.193,A -85,B 0,C 180,E1 -885.794,E2 -885.794} C_VEL
LIN {X 0,Y 601.391,Z 356.202,A -85,B 0,C 180,E1 -888.541,E2 -888.541} C_VEL
LIN {X 0,Y 601.361,Z 356.196,A -85,B 0,C 180,E1 -891.261,E2 -891.261} C_VEL
LIN {X 0,Y 601.367,Z 356.197,A -85,B 0,C 180,E1 -893.963,E2 -893.963} C_VEL
LIN {X 0,Y 601.409,Z 356.199,A -85,B 0,C 180,E1 -896.65,E2 -896.65} C_VEL
LIN {X 0,Y 601.35,Z 356.197,A -85,B 0,C 180,E1 -899.33,E2 -899.33} C_VEL
LIN {X 0,Y 601.362,Z 356.195,A -85,B 0,C 180,E1 -901.339,E2 -901.339} C_VEL
LIN {X 0,Y 601.34,Z 356.199,A -85,B 0,C 180,E1 -903.35,E2 -903.35} C_VEL
LIN {X 0,Y 601.369,Z 356.195,A -85,B 0,C 180,E1 -905.365,E2 -905.365} C_VEL
LIN {X 0,Y 601.35,Z 356.197,A -85,B 0,C 180,E1 -907.386,E2 -907.386} C_VEL
LIN {X 0,Y 601.358,Z 356.196,A -85,B 0,C 180,E1 -909.467,E2 -909.467} C_VEL
LIN {X 0,Y 601.38,Z 356.195,A -85,B 0,C 180,E1 -912.143,E2 -912.143} C_VEL
LIN {X 0,Y 601.376,Z 356.196,A -85,B 0,C 180,E1 -912.386,E2 -912.386} C_VEL
LIN {X 0,Y 600.72,Z 356.283,A -85,B 0,C 180,E1 -912.946,E2 -912.946} C_VEL
LIN {X 0,Y 597.874,Z 356.637,A -85,B 0,C 180,E1 -913.854,E2 -913.854} C_VEL
LIN {X 0,Y 595.457,Z 356.941,A -85,B 0,C 180,E1 -914.584,E2 -914.584} C_VEL
LIN {X 0,Y 594.411,Z 357.064,A -85,B 0,C 180,E1 -915.147,E2 -915.147} C_VEL
LIN {X 0,Y 594.322,Z 357.073,A -85,B 0,C 180,E1 -915.338,E2 -915.338} C_VEL
LIN {X 0,Y 594.359,Z 357.07,A -85,B 0,C 180,E1 -917.194,E2 -917.194} C_VEL
LIN {X 0,Y 594.34,Z 357.072,A -85,B 0,C 180,E1 -920.055,E2 -920.055} C_VEL
LIN {X 0,Y 594.333,Z 357.077,A -85,B 0,C 180,E1 -922.969,E2 -922.969} C_VEL
LIN {X 0,Y 594.304,Z 357.077,A -85,B 0,C 180,E1 -925.196,E2 -925.196} C_VEL
LIN {X 0,Y 594.327,Z 357.072,A -85,B 0,C 180,E1 -927.519,E2 -927.519} C_VEL
LIN {X 0,Y 594.316,Z 357.073,A -85,B 0,C 180,E1 -929.78,E2 -929.78} C_VEL
LIN {X 0,Y 594.341,Z 357.072,A -85,B 0,C 180,E1 -932.149,E2 -932.149} C_VEL
LIN {X 0,Y 594.363,Z 357.075,A -85,B 0,C 180,E1 -934.581,E2 -934.581} C_VEL
LIN {X 0,Y 594.337,Z 357.069,A -85,B 0,C 180,E1 -937.604,E2 -937.604} C_VEL
LIN {X 0,Y 594.316,Z 357.073,A -85,B 0,C 180,E1 -939.77,E2 -939.77} C_VEL
LIN {X 0,Y 594.322,Z 357.075,A -85,B 0,C 180,E1 -942.38,E2 -942.38} C_VEL
LIN {X 0,Y 594.304,Z 357.079,A -85,B 0,C 180,E1 -945.197,E2 -945.197} C_VEL
LIN {X 0,Y 594.316,Z 357.074,A -85,B 0,C 180,E1 -947.622,E2 -947.622} C_VEL
LIN {X 0,Y 594.343,Z 357.072,A -85,B 0,C 180,E1 -950.319,E2 -950.319} C_VEL
LIN {X 0,Y 594.364,Z 357.077,A -85,B 0,C 180,E1 -952.914,E2 -952.914} C_VEL
LIN {X 0,Y 594.341,Z 357.068,A -85,B 0,C 180,E1 -955.867,E2 -955.867} C_VEL
LIN {X 0,Y 594.336,Z 357.08,A -85,B 0,C 180,E1 -958.649,E2 -958.649} C_VEL
LIN {X 0,Y 594.358,Z 357.241,A -85,B 0,C 180,E1 -960.181,E2 -960.181} C_VEL
LIN {X 0,Y 595.435,Z 360.9,A -85,B 0,C 180,E1 -960.63,E2 -960.63} C_VEL
LIN {X 0,Y 595.635,Z 367.275,A -85,B 0,C 180,E1 -961.263,E2 -961.263} C_VEL
LIN {X 0,Y 595.373,Z 396.997,A -85,B 0,C 180,E1 -964.104,E2 -964.104} C_VEL
LIN {X 0,Y 595.137,Z 426.722,A -85,B 0,C 180,E1 -966.882,E2 -966.882} C_VEL
LIN {X 0,Y 594.937,Z 456.447,A -85,B 0,C 180,E1 -969.607,E2 -969.607} C_VEL
LIN {X 0,Y 594.887,Z 473.462,A -85,B 0,C 180,E1 -971.119,E2 -971.119} C_VEL
LIN {X 0,Y 595.315,Z 478.429,A -85,B 0,C 180,E1 -971.208,E2 -971.208} C_VEL
LIN {X 0,Y 595.083,Z 641.103,A -85,B 0,C 180,E1 -973.24,E2 -973.24} C_VEL
LIN {X 0,Y 595.024,Z 656.698,A -85,B 0,C 180,E1 -973.578,E2 -973.578} C_VEL
LIN {X 0,Y 594.933,Z 672.042,A -85,B 0,C 180,E1 -974.06,E2 -974.06} C_VEL
LIN {X 0,Y 594.835,Z 686.711,A -85,B 0,C 180,E1 -974.672,E2 -974.672} C_VEL
LIN {X 0,Y 594.742,Z 700.008,A -85,B 0,C 180,E1 -975.371,E2 -975.371} C_VEL
LIN {X 0,Y 594.669,Z 713.003,A -85,B 0,C 180,E1 -976.203,E2 -976.203} C_VEL
LIN {X 0,Y 594.551,Z 725.862,A -85,B 0,C 180,E1 -977.196,E2 -977.196} C_VEL
LIN {X 0,Y 594.467,Z 737.067,A -85,B 0,C 180,E1 -978.234,E2 -978.234} C_VEL
LIN {X 0,Y 594.412,Z 747.958,A -85,B 0,C 180,E1 -979.441,E2 -979.441} C_VEL
LIN {X 0,Y 594.356,Z 756.997,A -85,B 0,C 180,E1 -980.644,E2 -980.644} C_VEL
LIN {X 0,Y 594.325,Z 764.496,A -85,B 0,C 180,E1 -981.843,E2 -981.843} C_VEL
LIN {X 0,Y 594.275,Z 771.499,A -85,B 0,C 180,E1 -983.209,E2 -983.209} C_VEL
LIN {X 0,Y 594.272,Z 777.004,A -85,B 0,C 180,E1 -984.572,E2 -984.572} C_VEL
LIN {X 0,Y 594.254,Z 781.174,A -85,B 0,C 180,E1 -985.932,E2 -985.932} C_VEL
LIN {X 0,Y 594.221,Z 784.113,A -85,B 0,C 180,E1 -987.289,E2 -987.289} C_VEL
LIN {X 0,Y 594.244,Z 785.882,A -85,B 0,C 180,E1 -988.646,E2 -988.646} C_VEL
LIN {X 0,Y 594.234,Z 786.496,A -85,B 0,C 180,E1 -990.001,E2 -990.001} C_VEL
LIN {X 0,Y 594.246,Z 785.943,A -85,B 0,C 180,E1 -991.356,E2 -991.356} C_VEL
LIN {X 0,Y 594.223,Z 784.256,A -85,B 0,C 180,E1 -992.713,E2 -992.713} C_VEL
LIN {X 0,Y 594.254,Z 781.403,A -85,B 0,C 180,E1 -994.07,E2 -994.07} C_VEL
LIN {X 0,Y 594.272,Z 777.323,A -85,B 0,C 180,E1 -995.43,E2 -995.43} C_VEL
LIN {X 0,Y 594.278,Z 771.909,A -85,B 0,C 180,E1 -996.793,E2 -996.793} C_VEL
LIN {X 0,Y 594.314,Z 765.007,A -85,B 0,C 180,E1 -998.159,E2 -998.159} C_VEL
LIN {X 0,Y 594.339,Z 756.408,A -85,B 0,C 180,E1 -999.53,E2 -999.53} C_VEL
LIN {X 0,Y 594.401,Z 747.252,A -85,B 0,C 180,E1 -1000.733,E2 -1000.733} C_VEL
LIN {X 0,Y 594.467,Z 736.206,A -85,B 0,C 180,E1 -1001.941,E2 -1001.941} C_VEL
LIN {X 0,Y 594.56,Z 724.826,A -85,B 0,C 180,E1 -1002.98,E2 -1002.98} C_VEL
LIN {X 0,Y 594.661,Z 712.442,A -85,B 0,C 180,E1 -1003.926,E2 -1003.926} C_VEL
LIN {X 0,Y 594.723,Z 700.015,A -85,B 0,C 180,E1 -1004.719,E2 -1004.719} C_VEL
LIN {X 0,Y 594.855,Z 686.714,A -85,B 0,C 180,E1 -1005.417,E2 -1005.417} C_VEL
LIN {X 0,Y 594.903,Z 672.033,A -85,B 0,C 180,E1 -1006.031,E2 -1006.031} C_VEL
LIN {X 0,Y 595.038,Z 656.846,A -85,B 0,C 180,E1 -1006.508,E2 -1006.508} C_VEL
LIN {X 0,Y 595.083,Z 642.297,A -85,B 0,C 180,E1 -1006.829,E2 -1006.829} C_VEL
LIN {X 0,Y 595.156,Z 598.577,A -85,B 0,C 180,E1 -1007.393,E2 -1007.393} C_VEL
LIN {X 0,Y 595.172,Z 475.267,A -85,B 0,C 180,E1 -1008.926,E2 -1008.926} C_VEL
LIN {X 0,Y 594.843,Z 472.97,A -85,B 0,C 180,E1 -1008.999,E2 -1008.999} C_VEL
LIN {X 0,Y 595.038,Z 443.531,A -85,B 0,C 180,E1 -1011.661,E2 -1011.661} C_VEL
LIN {X 0,Y 595.286,Z 411.49,A -85,B 0,C 180,E1 -1014.623,E2 -1014.623} C_VEL
LIN {X 0,Y 595.533,Z 380.216,A -85,B 0,C 180,E1 -1017.581,E2 -1017.581} C_VEL
LIN {X 0,Y 595.665,Z 362.135,A -85,B 0,C 180,E1 -1019.327,E2 -1019.327} C_VEL
LIN {X 0,Y 594.349,Z 357.25,A -85,B 0,C 180,E1 -1019.907,E2 -1019.907} C_VEL
LIN {X 0,Y 594.329,Z 357.074,A -85,B 0,C 180,E1 -1022.15,E2 -1022.15} C_VEL
LIN {X 0,Y 594.298,Z 357.076,A -85,B 0,C 180,E1 -1024.586,E2 -1024.586} C_VEL
LIN {X 0,Y 594.35,Z 357.073,A -85,B 0,C 180,E1 -1027.603,E2 -1027.603} C_VEL
LIN {X 0,Y 594.316,Z 357.075,A -85,B 0,C 180,E1 -1030.572,E2 -1030.572} C_VEL
LIN {X 0,Y 594.341,Z 357.079,A -85,B 0,C 180,E1 -1033.303,E2 -1033.303} C_VEL
LIN {X 0,Y 594.316,Z 357.072,A -85,B 0,C 180,E1 -1036.167,E2 -1036.167} C_VEL
LIN {X 0,Y 594.36,Z 357.077,A -85,B 0,C 180,E1 -1039.181,E2 -1039.181} C_VEL
LIN {X 0,Y 594.306,Z 357.075,A -85,B 0,C 180,E1 -1042.053,E2 -1042.053} C_VEL
LIN {X 0,Y 594.324,Z 357.075,A -85,B 0,C 180,E1 -1044.681,E2 -1044.681} C_VEL
LIN {X 0,Y 594.344,Z 357.079,A -85,B 0,C 180,E1 -1047.095,E2 -1047.095} C_VEL
LIN {X 0,Y 594.349,Z 357.072,A -85,B 0,C 180,E1 -1049.679,E2 -1049.679} C_VEL
LIN {X 0,Y 594.332,Z 357.073,A -85,B 0,C 180,E1 -1051.771,E2 -1051.771} C_VEL
LIN {X 0,Y 594.342,Z 357.07,A -85,B 0,C 180,E1 -1054.054,E2 -1054.054} C_VEL
LIN {X 0,Y 594.349,Z 357.07,A -85,B 0,C 180,E1 -1056.294,E2 -1056.294} C_VEL
LIN {X 0,Y 594.404,Z 357.072,A -85,B 0,C 180,E1 -1059.224,E2 -1059.224} C_VEL
LIN {X 0,Y 594.406,Z 357.315,A -85,B 0,C 180,E1 -1060.967,E2 -1060.967} C_VEL
LIN {X 0,Y 594.488,Z 367.466,A -85,B 0,C 180,E1 -1062.632,E2 -1062.632} C_VEL
LIN {X 0,Y 594.481,Z 375.299,A -85,B 0,C 180,E1 -1063.87,E2 -1063.87} C_VEL
LIN {X 0,Y 594.853,Z 377.65,A -85,B 0,C 180,E1 -1063.948,E2 -1063.948} C_VEL
LIN {X 0,Y 594.887,Z 511.851,A -85,B 0,C 180,E1 -1065.613,E2 -1065.613} C_VEL
LIN {X 0,Y 594.843,Z 525.831,A -85,B 0,C 180,E1 -1065.925,E2 -1065.925} C_VEL
LIN {X 0,Y 594.773,Z 539.701,A -85,B 0,C 180,E1 -1066.374,E2 -1066.374} C_VEL
LIN {X 0,Y 594.682,Z 552.748,A -85,B 0,C 180,E1 -1066.937,E2 -1066.937} C_VEL
LIN {X 0,Y 594.596,Z 565.373,A -85,B 0,C 180,E1 -1067.629,E2 -1067.629} C_VEL
LIN {X 0,Y 594.519,Z 578.068,A -85,B 0,C 180,E1 -1068.496,E2 -1068.496} C_VEL
LIN {X 0,Y 594.449,Z 589.357,A -85,B 0,C 180,E1 -1069.441,E2 -1069.441} C_VEL
LIN {X 0,Y 594.371,Z 599.459,A -85,B 0,C 180,E1 -1070.471,E2 -1070.471} C_VEL
LIN {X 0,Y 594.324,Z 607.844,A -85,B 0,C 180,E1 -1071.5,E2 -1071.5} C_VEL
LIN {X 0,Y 594.304,Z 615.866,A -85,B 0,C 180,E1 -1072.696,E2 -1072.696} C_VEL
LIN {X 0,Y 594.279,Z 622.322,A -85,B 0,C 180,E1 -1073.89,E2 -1073.89} C_VEL
LIN {X 0,Y 594.235,Z 628.043,A -85,B 0,C 180,E1 -1075.251,E2 -1075.251} C_VEL
LIN {X 0,Y 594.26,Z 632.204,A -85,B 0,C 180,E1 -1076.61,E2 -1076.61} C_VEL
LIN {X 0,Y 594.239,Z 634.929,A -85,B 0,C 180,E1 -1077.967,E2 -1077.967} C_VEL
LIN {X 0,Y 594.235,Z 636.3,A -85,B 0,C 180,E1 -1079.322,E2 -1079.322} C_VEL
LIN {X 0,Y 594.235,Z 636.356,A -85,B 0,C 180,E1 -1080.678,E2 -1080.678} C_VEL
LIN {X 0,Y 594.237,Z 635.071,A -85,B 0,C 180,E1 -1082.033,E2 -1082.033} C_VEL
LIN {X 0,Y 594.26,Z 632.434,A -85,B 0,C 180,E1 -1083.39,E2 -1083.39} C_VEL
LIN {X 0,Y 594.236,Z 628.368,A -85,B 0,C 180,E1 -1084.749,E2 -1084.749} C_VEL
LIN {X 0,Y 594.28,Z 622.748,A -85,B 0,C 180,E1 -1086.11,E2 -1086.11} C_VEL
LIN {X 0,Y 594.304,Z 616.401,A -85,B 0,C 180,E1 -1087.303,E2 -1087.303} C_VEL
LIN {X 0,Y 594.325,Z 608.505,A -85,B 0,C 180,E1 -1088.5,E2 -1088.5} C_VEL
LIN {X 0,Y 594.356,Z 600.252,A -85,B 0,C 180,E1 -1089.529,E2 -1089.529} C_VEL
LIN {X 0,Y 594.449,Z 590.313,A -85,B 0,C 180,E1 -1090.559,E2 -1090.559} C_VEL
LIN {X 0,Y 594.492,Z 579.154,A -85,B 0,C 180,E1 -1091.513,E2 -1091.513} C_VEL
LIN {X 0,Y 594.581,Z 566.843,A -85,B 0,C 180,E1 -1092.371,E2 -1092.371} C_VEL
LIN {X 0,Y 594.642,Z 554.557,A -85,B 0,C 180,E1 -1093.064,E2 -1093.064} C_VEL
LIN {X 0,Y 594.717,Z 540.887,A -85,B 0,C 180,E1 -1093.671,E2 -1093.671} C_VEL
LIN {X 0,Y 594.8,Z 526.433,A -85,B 0,C 180,E1 -1094.149,E2 -1094.149} C_VEL
LIN {X 0,Y 594.864,Z 511.971,A -85,B 0,C 180,E1 -1094.474,E2 -1094.474} C_VEL
LIN {X 0,Y 594.874,Z 377.696,A -85,B 0,C 180,E1 -1096.141,E2 -1096.141} C_VEL
LIN {X 0,Y 594.48,Z 375.316,A -85,B 0,C 180,E1 -1096.218,E2 -1096.218} C_VEL
LIN {X 0,Y 594.526,Z 358.165,A -85,B 0,C 180,E1 -1098.968,E2 -1098.968} C_VEL
LIN {X 0,Y 594.396,Z 357.12,A -85,B 0,C 180,E1 -1099.217,E2 -1099.217} C_VEL
LIN {X 0,Y 594.362,Z 357.071,A -85,B 0,C 180,E1 -1101.503,E2 -1101.503} C_VEL
LIN {X 0,Y 594.392,Z 357.07,A -85,B 0,C 180,E1 -1104.446,E2 -1104.446} C_VEL
LIN {X 0,Y 594.384,Z 357.075,A -85,B 0,C 180,E1 -1106.7,E2 -1106.7} C_VEL
LIN {X 0,Y 594.385,Z 357.071,A -85,B 0,C 180,E1 -1108.998,E2 -1108.998} C_VEL
LIN {X 0,Y 594.38,Z 357.066,A -85,B 0,C 180,E1 -1111.642,E2 -1111.642} C_VEL
LIN {X 0,Y 594.38,Z 357.076,A -85,B 0,C 180,E1 -1114.58,E2 -1114.58} C_VEL
LIN {X 0,Y 594.389,Z 357.065,A -85,B 0,C 180,E1 -1117.608,E2 -1117.608} C_VEL
LIN {X 0,Y 594.365,Z 357.075,A -85,B 0,C 180,E1 -1120.567,E2 -1120.567} C_VEL
LIN {X 0,Y 594.353,Z 357.07,A -85,B 0,C 180,E1 -1123.301,E2 -1123.301} C_VEL
LIN {X 0,Y 594.347,Z 357.08,A -85,B 0,C 180,E1 -1126.163,E2 -1126.163} C_VEL
LIN {X 0,Y 594.367,Z 357.072,A -85,B 0,C 180,E1 -1128.534,E2 -1128.534} C_VEL
LIN {X 0,Y 594.364,Z 357.069,A -85,B 0,C 180,E1 -1131.298,E2 -1131.298} C_VEL
LIN {X 0,Y 594.343,Z 357.077,A -85,B 0,C 180,E1 -1133.754,E2 -1133.754} C_VEL
LIN {X 0,Y 594.342,Z 357.077,A -85,B 0,C 180,E1 -1136.236,E2 -1136.236} C_VEL
LIN {X 0,Y 594.31,Z 357.077,A -85,B 0,C 180,E1 -1138.645,E2 -1138.645} C_VEL
LIN {X 0,Y 594.349,Z 357.212,A -85,B 0,C 180,E1 -1141.058,E2 -1141.058} C_VEL
LIN {X 0,Y 595.273,Z 360.42,A -85,B 0,C 180,E1 -1141.434,E2 -1141.434} C_VEL
LIN {X 0,Y 595.697,Z 362.571,A -85,B 0,C 180,E1 -1141.649,E2 -1141.649} C_VEL
LIN {X 0,Y 595.438,Z 393.76,A -85,B 0,C 180,E1 -1144.386,E2 -1144.386} C_VEL
LIN {X 0,Y 595.184,Z 426.779,A -85,B 0,C 180,E1 -1147.221,E2 -1147.221} C_VEL
LIN {X 0,Y 594.971,Z 459.365,A -85,B 0,C 180,E1 -1149.966,E2 -1149.966} C_VEL
LIN {X 0,Y 594.924,Z 472.703,A -85,B 0,C 180,E1 -1151.063,E2 -1151.063} C_VEL
LIN {X 0,Y 595.299,Z 477.77,A -85,B 0,C 180,E1 -1151.155,E2 -1151.155} C_VEL
LIN {X 0,Y 595.104,Z 640.937,A -85,B 0,C 180,E1 -1153.192,E2 -1153.192} C_VEL
LIN {X 0,Y 595.007,Z 656.683,A -85,B 0,C 180,E1 -1153.531,E2 -1153.531} C_VEL
LIN {X 0,Y 594.934,Z 672.026,A -85,B 0,C 180,E1 -1154.014,E2 -1154.014} C_VEL
LIN {X 0,Y 594.858,Z 685.74,A -85,B 0,C 180,E1 -1154.583,E2 -1154.583} C_VEL
LIN {X 0,Y 594.733,Z 699.219,A -85,B 0,C 180,E1 -1155.281,E2 -1155.281} C_VEL
LIN {X 0,Y 594.682,Z 711.781,A -85,B 0,C 180,E1 -1156.074,E2 -1156.074} C_VEL
LIN {X 0,Y 594.56,Z 724.276,A -85,B 0,C 180,E1 -1157.02,E2 -1157.02} C_VEL
LIN {X 0,Y 594.466,Z 735.739,A -85,B 0,C 180,E1 -1158.059,E2 -1158.059} C_VEL
LIN {X 0,Y 594.389,Z 745.381,A -85,B 0,C 180,E1 -1159.094,E2 -1159.094} C_VEL
LIN {X 0,Y 594.367,Z 754.848,A -85,B 0,C 180,E1 -1160.299,E2 -1160.299} C_VEL
LIN {X 0,Y 594.311,Z 762.724,A -85,B 0,C 180,E1 -1161.499,E2 -1161.499} C_VEL
LIN {X 0,Y 594.293,Z 770.083,A -85,B 0,C 180,E1 -1162.866,E2 -1162.866} C_VEL
LIN {X 0,Y 594.296,Z 775.921,A -85,B 0,C 180,E1 -1164.23,E2 -1164.23} C_VEL
LIN {X 0,Y 594.232,Z 779.38,A -85,B 0,C 180,E1 -1165.25,E2 -1165.25} C_VEL
LIN {X 0,Y 594.257,Z 782.884,A -85,B 0,C 180,E1 -1166.609,E2 -1166.609} C_VEL
LIN {X 0,Y 594.238,Z 785.191,A -85,B 0,C 180,E1 -1167.966,E2 -1167.966} C_VEL
LIN {X 0,Y 594.237,Z 786.35,A -85,B 0,C 180,E1 -1169.321,E2 -1169.321} C_VEL
LIN {X 0,Y 594.237,Z 786.35,A -85,B 0,C 180,E1 -1170.677,E2 -1170.677} C_VEL
LIN {X 0,Y 594.238,Z 785.194,A -85,B 0,C 180,E1 -1172.032,E2 -1172.032} C_VEL
LIN {X 0,Y 594.257,Z 782.889,A -85,B 0,C 180,E1 -1173.389,E2 -1173.389} C_VEL
LIN {X 0,Y 594.232,Z 779.387,A -85,B 0,C 180,E1 -1174.748,E2 -1174.748} C_VEL
LIN {X 0,Y 594.275,Z 774.612,A -85,B 0,C 180,E1 -1176.109,E2 -1176.109} C_VEL
LIN {X 0,Y 594.296,Z 768.432,A -85,B 0,C 180,E1 -1177.473,E2 -1177.473} C_VEL
LIN {X 0,Y 594.33,Z 760.661,A -85,B 0,C 180,E1 -1178.842,E2 -1178.842} C_VEL
LIN {X 0,Y 594.386,Z 752.379,A -85,B 0,C 180,E1 -1180.043,E2 -1180.043} C_VEL
LIN {X 0,Y 594.432,Z 742.565,A -85,B 0,C 180,E1 -1181.23,E2 -1181.23} C_VEL
LIN {X 0,Y 594.53,Z 732.204,A -85,B 0,C 180,E1 -1182.284,E2 -1182.284} C_VEL
LIN {X 0,Y 594.581,Z 720.031,A -85,B 0,C 180,E1 -1183.325,E2 -1183.325} C_VEL
LIN {X 0,Y 594.691,Z 708.092,A -85,B 0,C 180,E1 -1184.177,E2 -1184.177} C_VEL
LIN {X 0,Y 594.779,Z 694.549,A -85,B 0,C 180,E1 -1184.979,E2 -1184.979} C_VEL
LIN {X 0,Y 594.902,Z 679.87,A -85,B 0,C 180,E1 -1185.677,E2 -1185.677} C_VEL
LIN {X 0,Y 594.965,Z 665.652,A -85,B 0,C 180,E1 -1186.203,E2 -1186.203} C_VEL
LIN {X 0,Y 595.053,Z 651.079,A -85,B 0,C 180,E1 -1186.604,E2 -1186.604} C_VEL
LIN {X 0,Y 595.083,Z 635.559,A -85,B 0,C 180,E1 -1186.888,E2 -1186.888} C_VEL
LIN {X 0,Y 595.266,Z 475.135,A -85,B 0,C 180,E1 -1188.879,E2 -1188.879} C_VEL
LIN {X 0,Y 594.89,Z 472.533,A -85,B 0,C 180,E1 -1188.948,E2 -1188.948} C_VEL
LIN {X 0,Y 595.123,Z 437.882,A -85,B 0,C 180,E1 -1191.837,E2 -1191.837} C_VEL
LIN {X 0,Y 595.356,Z 404.053,A -85,B 0,C 180,E1 -1194.723,E2 -1194.723} C_VEL
LIN {X 0,Y 595.632,Z 371.116,A -85,B 0,C 180,E1 -1197.595,E2 -1197.595} C_VEL
LIN {X 0,Y 595.638,Z 361.522,A -85,B 0,C 180,E1 -1198.448,E2 -1198.448} C_VEL
LIN {X 0,Y 594.343,Z 357.218,A -85,B 0,C 180,E1 -1198.941,E2 -1198.941} C_VEL
LIN {X 0,Y 594.317,Z 357.074,A -85,B 0,C 180,E1 -1201.352,E2 -1201.352} C_VEL
LIN {X 0,Y 594.348,Z 357.079,A -85,B 0,C 180,E1 -1204.134,E2 -1204.134} C_VEL
LIN {X 0,Y 594.311,Z 357.075,A -85,B 0,C 180,E1 -1207.09,E2 -1207.09} C_VEL
LIN {X 0,Y 594.328,Z 357.074,A -85,B 0,C 180,E1 -1209.769,E2 -1209.769} C_VEL
LIN {X 0,Y 594.353,Z 357.079,A -85,B 0,C 180,E1 -1212.375,E2 -1212.375} C_VEL
LIN {X 0,Y 594.301,Z 357.075,A -85,B 0,C 180,E1 -1215.195,E2 -1215.195} C_VEL
LIN {X 0,Y 594.352,Z 357.074,A -85,B 0,C 180,E1 -1218.153,E2 -1218.153} C_VEL
LIN {X 0,Y 594.34,Z 357.07,A -85,B 0,C 180,E1 -1221.192,E2 -1221.192} C_VEL
LIN {X 0,Y 594.325,Z 357.072,A -85,B 0,C 180,E1 -1223.754,E2 -1223.754} C_VEL
LIN {X 0,Y 594.358,Z 357.073,A -85,B 0,C 180,E1 -1226.237,E2 -1226.237} C_VEL
LIN {X 0,Y 594.344,Z 357.076,A -85,B 0,C 180,E1 -1228.648,E2 -1228.648} C_VEL
LIN {X 0,Y 594.353,Z 357.069,A -85,B 0,C 180,E1 -1231.044,E2 -1231.044} C_VEL
LIN {X 0,Y 594.354,Z 357.073,A -85,B 0,C 180,E1 -1234.055,E2 -1234.055} C_VEL
LIN {X 0,Y 594.331,Z 357.073,A -85,B 0,C 180,E1 -1237.031,E2 -1237.031} C_VEL
LIN {X 0,Y 594.335,Z 357.073,A -85,B 0,C 180,E1 -1239.945,E2 -1239.945} C_VEL
LIN {X 0,Y 594.311,Z 357.079,A -85,B 0,C 180,E1 -1242.804,E2 -1242.804} C_VEL
LIN {X 0,Y 594.333,Z 357.07,A -85,B 0,C 180,E1 -1245.622,E2 -1245.622} C_VEL
LIN {X 0,Y 594.356,Z 357.077,A -85,B 0,C 180,E1 -1248.404,E2 -1248.404} C_VEL
LIN {X 0,Y 594.334,Z 357.072,A -85,B 0,C 180,E1 -1251.157,E2 -1251.157} C_VEL
LIN {X 0,Y 594.319,Z 357.074,A -85,B 0,C 180,E1 -1253.891,E2 -1253.891} C_VEL
LIN {X 0,Y 594.359,Z 357.078,A -85,B 0,C 180,E1 -1256.611,E2 -1256.611} C_VEL
LIN {X 0,Y 594.306,Z 357.075,A -85,B 0,C 180,E1 -1259.322,E2 -1259.322} C_VEL
LIN {X 0,Y 594.319,Z 357.072,A -85,B 0,C 180,E1 -1261.355,E2 -1261.355} C_VEL
LIN {X 0,Y 594.294,Z 357.076,A -85,B 0,C 180,E1 -1263.39,E2 -1263.39} C_VEL
LIN {X 0,Y 594.336,Z 357.07,A -85,B 0,C 180,E1 -1265.428,E2 -1265.428} C_VEL
LIN {X 0,Y 594.323,Z 357.072,A -85,B 0,C 180,E1 -1267.474,E2 -1267.474} C_VEL
LIN {X 0,Y 594.311,Z 357.074,A -85,B 0,C 180,E1 -1269.53,E2 -1269.53} C_VEL
LIN {X 0,Y 594.359,Z 357.071,A -85,B 0,C 180,E1 -1272.289,E2 -1272.289} C_VEL
LIN {X 0,Y 594.34,Z 357.073,A -85,B 0,C 180,E1 -1275.079,E2 -1275.079} C_VEL
LIN {X 0,Y 594.322,Z 357.073,A -85,B 0,C 180,E1 -1275.338,E2 -1275.338} C_VEL
LIN {X 0,Y 593.639,Z 357.158,A -85,B 0,C 180,E1 -1275.904,E2 -1275.904} C_VEL
LIN {X 0,Y 590.766,Z 357.523,A -85,B 0,C 180,E1 -1276.822,E2 -1276.822} C_VEL
LIN {X 0,Y 588.36,Z 357.819,A -85,B 0,C 180,E1 -1277.561,E2 -1277.561} C_VEL
LIN {X 0,Y 587.348,Z 357.943,A -85,B 0,C 180,E1 -1278.131,E2 -1278.131} C_VEL
LIN {X 0,Y 587.277,Z 357.952,A -85,B 0,C 180,E1 -1278.324,E2 -1278.324} C_VEL
LIN {X 0,Y 587.315,Z 357.949,A -85,B 0,C 180,E1 -1281.038,E2 -1281.038} C_VEL
LIN {X 0,Y 587.279,Z 357.951,A -85,B 0,C 180,E1 -1284.009,E2 -1284.009} C_VEL
LIN {X 0,Y 587.269,Z 357.954,A -85,B 0,C 180,E1 -1286.282,E2 -1286.282} C_VEL
LIN {X 0,Y 587.325,Z 357.948,A -85,B 0,C 180,E1 -1289.133,E2 -1289.133} C_VEL
LIN {X 0,Y 587.299,Z 357.948,A -85,B 0,C 180,E1 -1291.832,E2 -1291.832} C_VEL
LIN {X 0,Y 587.324,Z 357.949,A -85,B 0,C 180,E1 -1294.347,E2 -1294.347} C_VEL
LIN {X 0,Y 587.292,Z 357.946,A -85,B 0,C 180,E1 -1297.612,E2 -1297.612} C_VEL
LIN {X 0,Y 587.284,Z 357.952,A -85,B 0,C 180,E1 -1300.257,E2 -1300.257} C_VEL
LIN {X 0,Y 587.276,Z 357.955,A -85,B 0,C 180,E1 -1303.116,E2 -1303.116} C_VEL
LIN {X 0,Y 587.276,Z 357.951,A -85,B 0,C 180,E1 -1306.047,E2 -1306.047} C_VEL
LIN {X 0,Y 587.298,Z 357.956,A -85,B 0,C 180,E1 -1308.929,E2 -1308.929} C_VEL
LIN {X 0,Y 587.29,Z 357.95,A -85,B 0,C 180,E1 -1311.52,E2 -1311.52} C_VEL
LIN {X 0,Y 587.245,Z 357.956,A -85,B 0,C 180,E1 -1314.099,E2 -1314.099} C_VEL
LIN {X 0,Y 587.298,Z 357.949,A -85,B 0,C 180,E1 -1316.603,E2 -1316.603} C_VEL
LIN {X 0,Y 587.296,Z 357.956,A -85,B 0,C 180,E1 -1319.497,E2 -1319.497} C_VEL
LIN {X 0,Y 587.348,Z 358.217,A -85,B 0,C 180,E1 -1319.932,E2 -1319.932} C_VEL
LIN {X 0,Y 588.978,Z 364.012,A -85,B 0,C 180,E1 -1320.584,E2 -1320.584} C_VEL
LIN {X 0,Y 588.779,Z 387.096,A -85,B 0,C 180,E1 -1322.835,E2 -1322.835} C_VEL
LIN {X 0,Y 588.514,Z 414.838,A -85,B 0,C 180,E1 -1325.483,E2 -1325.483} C_VEL
LIN {X 0,Y 588.213,Z 446.276,A -85,B 0,C 180,E1 -1328.421,E2 -1328.421} C_VEL
LIN {X 0,Y 588.016,Z 473.35,A -85,B 0,C 180,E1 -1330.885,E2 -1330.885} C_VEL
LIN {X 0,Y 588.597,Z 477.974,A -85,B 0,C 180,E1 -1330.979,E2 -1330.979} C_VEL
LIN {X 0,Y 588.311,Z 640.625,A -85,B 0,C 180,E1 -1333.033,E2 -1333.033} C_VEL
LIN {X 0,Y 588.226,Z 655.858,A -85,B 0,C 180,E1 -1333.36,E2 -1333.36} C_VEL
LIN {X 0,Y 588.119,Z 670.817,A -85,B 0,C 180,E1 -1333.826,E2 -1333.826} C_VEL
LIN {X 0,Y 587.989,Z 684.81,A -85,B 0,C 180,E1 -1334.4,E2 -1334.4} C_VEL
LIN {X 0,Y 587.82,Z 698.473,A -85,B 0,C 180,E1 -1335.106,E2 -1335.106} C_VEL
LIN {X 0,Y 587.744,Z 711.517,A -85,B 0,C 180,E1 -1335.933,E2 -1335.933} C_VEL
LIN {X 0,Y 587.581,Z 723.766,A -85,B 0,C 180,E1 -1336.866,E2 -1336.866} C_VEL
LIN {X 0,Y 587.467,Z 735.313,A -85,B 0,C 180,E1 -1337.917,E2 -1337.917} C_VEL
LIN {X 0,Y 587.366,Z 745.025,A -85,B 0,C 180,E1 -1338.964,E2 -1338.964} C_VEL
LIN {X 0,Y 587.31,Z 754.551,A -85,B 0,C 180,E1 -1340.183,E2 -1340.183} C_VEL
LIN {X 0,Y 587.239,Z 763.491,A -85,B 0,C 180,E1 -1341.571,E2 -1341.571} C_VEL
LIN {X 0,Y 587.215,Z 769.887,A -85,B 0,C 180,E1 -1342.782,E2 -1342.782} C_VEL
LIN {X 0,Y 587.225,Z 775.77,A -85,B 0,C 180,E1 -1344.162,E2 -1344.162} C_VEL
LIN {X 0,Y 587.134,Z 779.25,A -85,B 0,C 180,E1 -1345.195,E2 -1345.195} C_VEL
LIN {X 0,Y 587.179,Z 782.793,A -85,B 0,C 180,E1 -1346.57,E2 -1346.57} C_VEL
LIN {X 0,Y 587.139,Z 785.141,A -85,B 0,C 180,E1 -1347.943,E2 -1347.943} C_VEL
LIN {X 0,Y 587.135,Z 786.338,A -85,B 0,C 180,E1 -1349.315,E2 -1349.315} C_VEL
LIN {X 0,Y 587.136,Z 786.36,A -85,B 0,C 180,E1 -1350.687,E2 -1350.687} C_VEL
LIN {X 0,Y 587.14,Z 785.242,A -85,B 0,C 180,E1 -1352.059,E2 -1352.059} C_VEL
LIN {X 0,Y 587.181,Z 782.978,A -85,B 0,C 180,E1 -1353.432,E2 -1353.432} C_VEL
LIN {X 0,Y 587.134,Z 779.52,A -85,B 0,C 180,E1 -1354.807,E2 -1354.807} C_VEL
LIN {X 0,Y 587.182,Z 774.788,A -85,B 0,C 180,E1 -1356.185,E2 -1356.185} C_VEL
LIN {X 0,Y 587.23,Z 768.65,A -85,B 0,C 180,E1 -1357.566,E2 -1357.566} C_VEL
LIN {X 0,Y 587.266,Z 760.931,A -85,B 0,C 180,E1 -1358.951,E2 -1358.951} C_VEL
LIN {X 0,Y 587.353,Z 752.695,A -85,B 0,C 180,E1 -1360.166,E2 -1360.166} C_VEL
LIN {X 0,Y 587.4,Z 742.786,A -85,B 0,C 180,E1 -1361.386,E2 -1361.386} C_VEL
LIN {X 0,Y 587.501,Z 732.65,A -85,B 0,C 180,E1 -1362.436,E2 -1362.436} C_VEL
LIN {X 0,Y 587.621,Z 720.57,A -85,B 0,C 180,E1 -1363.488,E2 -1363.488} C_VEL
LIN {X 0,Y 587.761,Z 707.829,A -85,B 0,C 180,E1 -1364.411,E2 -1364.411} C_VEL
LIN {X 0,Y 587.874,Z 693.701,A -85,B 0,C 180,E1 -1365.25,E2 -1365.25} C_VEL
LIN {X 0,Y 588.048,Z 678.757,A -85,B 0,C 180,E1 -1365.956,E2 -1365.956} C_VEL
LIN {X 0,Y 588.152,Z 664.241,A -85,B 0,C 180,E1 -1366.488,E2 -1366.488} C_VEL
LIN {X 0,Y 588.264,Z 648.877,A -85,B 0,C 180,E1 -1366.898,E2 -1366.898} C_VEL
LIN {X 0,Y 588.333,Z 633.446,A -85,B 0,C 180,E1 -1367.164,E2 -1367.164} C_VEL
LIN {X 0,Y 588.581,Z 477.113,A -85,B 0,C 180,E1 -1369.122,E2 -1369.122} C_VEL
LIN {X 0,Y 588.008,Z 472.997,A -85,B 0,C 180,E1 -1369.226,E2 -1369.226} C_VEL
LIN {X 0,Y 588.23,Z 443.524,A -85,B 0,C 180,E1 -1371.924,E2 -1371.924} C_VEL
LIN {X 0,Y 588.528,Z 413.78,A -85,B 0,C 180,E1 -1374.707,E2 -1374.707} C_VEL
LIN {X 0,Y 588.9,Z 381.252,A -85,B 0,C 180,E1 -1377.817,E2 -1377.817} C_VEL
LIN {X 0,Y 589.068,Z 364.713,A -85,B 0,C 180,E1 -1379.432,E2 -1379.432} C_VEL
LIN {X 0,Y 587.299,Z 358.069,A -85,B 0,C 180,E1 -1380.193,E2 -1380.193} C_VEL
LIN {X 0,Y 587.301,Z 357.952,A -85,B 0,C 180,E1 -1382.582,E2 -1382.582} C_VEL
LIN {X 0,Y 587.246,Z 357.96,A -85,B 0,C 180,E1 -1385.531,E2 -1385.531} C_VEL
LIN {X 0,Y 587.278,Z 357.952,A -85,B 0,C 180,E1 -1387.831,E2 -1387.831} C_VEL
LIN {X 0,Y 587.276,Z 357.951,A -85,B 0,C 180,E1 -1390.258,E2 -1390.258} C_VEL
LIN {X 0,Y 587.283,Z 357.958,A -85,B 0,C 180,E1 -1393.115,E2 -1393.115} C_VEL
LIN {X 0,Y 587.273,Z 357.95,A -85,B 0,C 180,E1 -1396.045,E2 -1396.045} C_VEL
LIN {X 0,Y 587.295,Z 357.955,A -85,B 0,C 180,E1 -1398.93,E2 -1398.93} C_VEL
LIN {X 0,Y 587.292,Z 357.953,A -85,B 0,C 180,E1 -1401.518,E2 -1401.518} C_VEL
LIN {X 0,Y 587.269,Z 357.95,A -85,B 0,C 180,E1 -1404.098,E2 -1404.098} C_VEL
LIN {X 0,Y 587.296,Z 357.948,A -85,B 0,C 180,E1 -1406.601,E2 -1406.601} C_VEL
LIN {X 0,Y 587.305,Z 357.956,A -85,B 0,C 180,E1 -1409.032,E2 -1409.032} C_VEL
LIN {X 0,Y 587.299,Z 357.954,A -85,B 0,C 180,E1 -1411.402,E2 -1411.402} C_VEL
LIN {X 0,Y 587.297,Z 357.949,A -85,B 0,C 180,E1 -1413.832,E2 -1413.832} C_VEL
LIN {X 0,Y 587.302,Z 357.952,A -85,B 0,C 180,E1 -1416.74,E2 -1416.74} C_VEL
LIN {X 0,Y 587.317,Z 357.95,A -85,B 0,C 180,E1 -1419.695,E2 -1419.695} C_VEL
LIN {X 0,Y 587.354,Z 358.123,A -85,B 0,C 180,E1 -1420.857,E2 -1420.857} C_VEL
LIN {X 0,Y 587.549,Z 364.18,A -85,B 0,C 180,E1 -1421.88,E2 -1421.88} C_VEL
LIN {X 0,Y 587.491,Z 375.321,A -85,B 0,C 180,E1 -1423.673,E2 -1423.673} C_VEL
LIN {X 0,Y 588.012,Z 378.431,A -85,B 0,C 180,E1 -1423.765,E2 -1423.765} C_VEL
LIN {X 0,Y 588.016,Z 511.885,A -85,B 0,C 180,E1 -1425.442,E2 -1425.442} C_VEL
LIN {X 0,Y 587.943,Z 526.221,A -85,B 0,C 180,E1 -1425.767,E2 -1425.767} C_VEL
LIN {X 0,Y 587.837,Z 539.726,A -85,B 0,C 180,E1 -1426.21,E2 -1426.21} C_VEL
LIN {X 0,Y 587.732,Z 552.769,A -85,B 0,C 180,E1 -1426.78,E2 -1426.78} C_VEL
LIN {X 0,Y 587.628,Z 565.389,A -85,B 0,C 180,E1 -1427.48,E2 -1427.48} C_VEL
LIN {X 0,Y 587.514,Z 576.884,A -85,B 0,C 180,E1 -1428.267,E2 -1428.267} C_VEL
LIN {X 0,Y 587.467,Z 587.435,A -85,B 0,C 180,E1 -1429.139,E2 -1429.139} C_VEL
LIN {X 0,Y 587.355,Z 597.914,A -85,B 0,C 180,E1 -1430.183,E2 -1430.183} C_VEL
LIN {X 0,Y 587.311,Z 606.567,A -85,B 0,C 180,E1 -1431.224,E2 -1431.224} C_VEL
LIN {X 0,Y 587.251,Z 614.84,A -85,B 0,C 180,E1 -1432.435,E2 -1432.435} C_VEL
LIN {X 0,Y 587.18,Z 621.469,A -85,B 0,C 180,E1 -1433.637,E2 -1433.637} C_VEL
LIN {X 0,Y 587.159,Z 626.784,A -85,B 0,C 180,E1 -1434.849,E2 -1434.849} C_VEL
LIN {X 0,Y 587.18,Z 630.314,A -85,B 0,C 180,E1 -1435.882,E2 -1435.882} C_VEL
LIN {X 0,Y 587.131,Z 633.743,A -85,B 0,C 180,E1 -1437.256,E2 -1437.256} C_VEL
LIN {X 0,Y 587.145,Z 635.778,A -85,B 0,C 180,E1 -1438.628,E2 -1438.628} C_VEL
LIN {X 0,Y 587.133,Z 636.496,A -85,B 0,C 180,E1 -1440,E2 -1440} C_VEL
LIN {X 0,Y 587.141,Z 635.88,A -85,B 0,C 180,E1 -1441.372,E2 -1441.372} C_VEL
LIN {X 0,Y 587.131,Z 633.924,A -85,B 0,C 180,E1 -1442.744,E2 -1442.744} C_VEL
LIN {X 0,Y 587.181,Z 630.584,A -85,B 0,C 180,E1 -1444.118,E2 -1444.118} C_VEL
LIN {X 0,Y 587.199,Z 625.764,A -85,B 0,C 180,E1 -1445.494,E2 -1445.494} C_VEL
LIN {X 0,Y 587.211,Z 619.301,A -85,B 0,C 180,E1 -1446.874,E2 -1446.874} C_VEL
LIN {X 0,Y 587.269,Z 612.104,A -85,B 0,C 180,E1 -1448.083,E2 -1448.083} C_VEL
LIN {X 0,Y 587.317,Z 603.177,A -85,B 0,C 180,E1 -1449.297,E2 -1449.297} C_VEL
LIN {X 0,Y 587.372,Z 593.839,A -85,B 0,C 180,E1 -1450.339,E2 -1450.339} C_VEL
LIN {X 0,Y 587.471,Z 583.599,A -85,B 0,C 180,E1 -1451.289,E2 -1451.289} C_VEL
LIN {X 0,Y 587.569,Z 572.105,A -85,B 0,C 180,E1 -1452.17,E2 -1452.17} C_VEL
LIN {X 0,Y 587.663,Z 559.471,A -85,B 0,C 180,E1 -1452.958,E2 -1452.958} C_VEL
LIN {X 0,Y 587.806,Z 546.197,A -85,B 0,C 180,E1 -1453.615,E2 -1453.615} C_VEL
LIN {X 0,Y 587.907,Z 532.213,A -85,B 0,C 180,E1 -1454.144,E2 -1454.144} C_VEL
LIN {X 0,Y 587.959,Z 517.618,A -85,B 0,C 180,E1 -1454.538,E2 -1454.538} C_VEL
LIN {X 0,Y 588.02,Z 502.889,A -85,B 0,C 180,E1 -1454.779,E2 -1454.779} C_VEL
LIN {X 0,Y 588.189,Z 379.442,A -85,B 0,C 180,E1 -1456.307,E2 -1456.307} C_VEL
LIN {X 0,Y 587.508,Z 375.634,A -85,B 0,C 180,E1 -1456.394,E2 -1456.394} C_VEL
LIN {X 0,Y 587.446,Z 373.505,A -85,B 0,C 180,E1 -1456.686,E2 -1456.686} C_VEL
LIN {X 0,Y 587.482,Z 358.927,A -85,B 0,C 180,E1 -1459.078,E2 -1459.078} C_VEL
LIN {X 0,Y 587.348,Z 358.02,A -85,B 0,C 180,E1 -1459.279,E2 -1459.279} C_VEL
LIN {X 0,Y 587.318,Z 357.948,A -85,B 0,C 180,E1 -1461.774,E2 -1461.774} C_VEL
LIN {X 0,Y 587.355,Z 357.951,A -85,B 0,C 180,E1 -1464.758,E2 -1464.758} C_VEL
LIN {X 0,Y 587.332,Z 357.95,A -85,B 0,C 180,E1 -1467.046,E2 -1467.046} C_VEL
LIN {X 0,Y 587.351,Z 357.943,A -85,B 0,C 180,E1 -1469.379,E2 -1469.379} C_VEL
LIN {X 0,Y 587.347,Z 357.943,A -85,B 0,C 180,E1 -1471.835,E2 -1471.835} C_VEL
LIN {X 0,Y 587.35,Z 357.949,A -85,B 0,C 180,E1 -1474.347,E2 -1474.347} C_VEL
LIN {X 0,Y 587.345,Z 357.943,A -85,B 0,C 180,E1 -1477.608,E2 -1477.608} C_VEL
LIN {X 0,Y 587.312,Z 357.955,A -85,B 0,C 180,E1 -1480.254,E2 -1480.254} C_VEL
LIN {X 0,Y 587.304,Z 357.948,A -85,B 0,C 180,E1 -1483.116,E2 -1483.116} C_VEL
LIN {X 0,Y 587.303,Z 357.956,A -85,B 0,C 180,E1 -1486.047,E2 -1486.047} C_VEL
LIN {X 0,Y 587.309,Z 357.948,A -85,B 0,C 180,E1 -1488.84,E2 -1488.84} C_VEL
LIN {X 0,Y 587.313,Z 357.949,A -85,B 0,C 180,E1 -1491.519,E2 -1491.519} C_VEL
LIN {X 0,Y 587.274,Z 357.96,A -85,B 0,C 180,E1 -1494.098,E2 -1494.098} C_VEL
LIN {X 0,Y 587.304,Z 357.95,A -85,B 0,C 180,E1 -1496.601,E2 -1496.601} C_VEL
LIN {X 0,Y 587.31,Z 357.954,A -85,B 0,C 180,E1 -1499.495,E2 -1499.495} C_VEL
LIN {X 0,Y 587.312,Z 358.187,A -85,B 0,C 180,E1 -1500.781,E2 -1500.781} C_VEL
LIN {X 0,Y 589.095,Z 364.722,A -85,B 0,C 180,E1 -1501.496,E2 -1501.496} C_VEL
LIN {X 0,Y 588.736,Z 395.911,A -85,B 0,C 180,E1 -1504.263,E2 -1504.263} C_VEL
LIN {X 0,Y 588.42,Z 428.91,A -85,B 0,C 180,E1 -1507.129,E2 -1507.129} C_VEL
LIN {X 0,Y 588.113,Z 461.516,A -85,B 0,C 180,E1 -1509.905,E2 -1509.905} C_VEL
LIN {X 0,Y 588.081,Z 472.677,A -85,B 0,C 180,E1 -1510.833,E2 -1510.833} C_VEL
LIN {X 0,Y 588.599,Z 477.586,A -85,B 0,C 180,E1 -1510.929,E2 -1510.929} C_VEL
LIN {X 0,Y 588.306,Z 641.254,A -85,B 0,C 180,E1 -1512.997,E2 -1512.997} C_VEL
LIN {X 0,Y 588.203,Z 656.683,A -85,B 0,C 180,E1 -1513.335,E2 -1513.335} C_VEL
LIN {X 0,Y 588.072,Z 672.025,A -85,B 0,C 180,E1 -1513.822,E2 -1513.822} C_VEL
LIN {X 0,Y 587.99,Z 685.742,A -85,B 0,C 180,E1 -1514.398,E2 -1514.398} C_VEL
LIN {X 0,Y 587.83,Z 699.221,A -85,B 0,C 180,E1 -1515.104,E2 -1515.104} C_VEL
LIN {X 0,Y 587.733,Z 712.104,A -85,B 0,C 180,E1 -1515.928,E2 -1515.928} C_VEL
LIN {X 0,Y 587.583,Z 724.277,A -85,B 0,C 180,E1 -1516.863,E2 -1516.863} C_VEL
LIN {X 0,Y 587.454,Z 735.739,A -85,B 0,C 180,E1 -1517.914,E2 -1517.914} C_VEL
LIN {X 0,Y 587.349,Z 745.382,A -85,B 0,C 180,E1 -1518.962,E2 -1518.962} C_VEL
LIN {X 0,Y 587.305,Z 754.849,A -85,B 0,C 180,E1 -1520.181,E2 -1520.181} C_VEL
LIN {X 0,Y 587.264,Z 762.724,A -85,B 0,C 180,E1 -1521.396,E2 -1521.396} C_VEL
LIN {X 0,Y 587.216,Z 770.083,A -85,B 0,C 180,E1 -1522.78,E2 -1522.78} C_VEL
LIN {X 0,Y 587.224,Z 775.921,A -85,B 0,C 180,E1 -1524.16,E2 -1524.16} C_VEL
LIN {X 0,Y 587.136,Z 779.381,A -85,B 0,C 180,E1 -1525.193,E2 -1525.193} C_VEL
LIN {X 0,Y 587.179,Z 782.884,A -85,B 0,C 180,E1 -1526.568,E2 -1526.568} C_VEL
LIN {X 0,Y 587.137,Z 785.191,A -85,B 0,C 180,E1 -1527.941,E2 -1527.941} C_VEL
LIN {X 0,Y 587.137,Z 786.349,A -85,B 0,C 180,E1 -1529.313,E2 -1529.313} C_VEL
LIN {X 0,Y 587.137,Z 786.35,A -85,B 0,C 180,E1 -1530.685,E2 -1530.685} C_VEL
LIN {X 0,Y 587.137,Z 785.194,A -85,B 0,C 180,E1 -1532.057,E2 -1532.057} C_VEL
LIN {X 0,Y 587.179,Z 782.89,A -85,B 0,C 180,E1 -1533.43,E2 -1533.43} C_VEL
LIN {X 0,Y 587.136,Z 779.387,A -85,B 0,C 180,E1 -1534.805,E2 -1534.805} C_VEL
LIN {X 0,Y 587.178,Z 774.612,A -85,B 0,C 180,E1 -1536.183,E2 -1536.183} C_VEL
LIN {X 0,Y 587.235,Z 768.431,A -85,B 0,C 180,E1 -1537.564,E2 -1537.564} C_VEL
LIN {X 0,Y 587.266,Z 760.66,A -85,B 0,C 180,E1 -1538.949,E2 -1538.949} C_VEL
LIN {X 0,Y 587.351,Z 752.379,A -85,B 0,C 180,E1 -1540.164,E2 -1540.164} C_VEL
LIN {X 0,Y 587.398,Z 742.406,A -85,B 0,C 180,E1 -1541.384,E2 -1541.384} C_VEL
LIN {X 0,Y 587.521,Z 732.203,A -85,B 0,C 180,E1 -1542.433,E2 -1542.433} C_VEL
LIN {X 0,Y 587.628,Z 720.031,A -85,B 0,C 180,E1 -1543.485,E2 -1543.485} C_VEL
LIN {X 0,Y 587.771,Z 707.075,A -85,B 0,C 180,E1 -1544.415,E2 -1544.415} C_VEL
LIN {X 0,Y 587.886,Z 692.893,A -85,B 0,C 180,E1 -1545.247,E2 -1545.247} C_VEL
LIN {X 0,Y 588.048,Z 678.828,A -85,B 0,C 180,E1 -1545.909,E2 -1545.909} C_VEL
LIN {X 0,Y 588.167,Z 664.337,A -85,B 0,C 180,E1 -1546.44,E2 -1546.44} C_VEL
LIN {X 0,Y 588.268,Z 649.248,A -85,B 0,C 180,E1 -1546.845,E2 -1546.845} C_VEL
LIN {X 0,Y 588.322,Z 634.056,A -85,B 0,C 180,E1 -1547.11,E2 -1547.11} C_VEL
LIN {X 0,Y 588.558,Z 476.116,A -85,B 0,C 180,E1 -1549.091,E2 -1549.091} C_VEL
LIN {X 0,Y 588.054,Z 472.472,A -85,B 0,C 180,E1 -1549.181,E2 -1549.181} C_VEL
LIN {X 0,Y 588.332,Z 438.957,A -85,B 0,C 180,E1 -1552.01,E2 -1552.01} C_VEL
LIN {X 0,Y 588.662,Z 405.953,A -85,B 0,C 180,E1 -1554.857,E2 -1554.857} C_VEL
LIN {X 0,Y 589.023,Z 372.134,A -85,B 0,C 180,E1 -1557.84,E2 -1557.84} C_VEL
LIN {X 0,Y 589.092,Z 364.748,A -85,B 0,C 180,E1 -1558.502,E2 -1558.502} C_VEL
LIN {X 0,Y 587.307,Z 358.196,A -85,B 0,C 180,E1 -1559.217,E2 -1559.217} C_VEL
LIN {X 0,Y 587.317,Z 357.947,A -85,B 0,C 180,E1 -1560.169,E2 -1560.169} C_VEL
LIN {X 0,Y 587.319,Z 357.947,A -85,B 0,C 180,E1 -1563.109,E2 -1563.109} C_VEL
LIN {X 0,Y 587.263,Z 357.957,A -85,B 0,C 180,E1 -1565.9,E2 -1565.9} C_VEL
LIN {X 0,Y 587.3,Z 357.955,A -85,B 0,C 180,E1 -1568.48,E2 -1568.48} C_VEL
LIN {X 0,Y 587.289,Z 357.949,A -85,B 0,C 180,E1 -1571.159,E2 -1571.159} C_VEL
LIN {X 0,Y 587.285,Z 357.954,A -85,B 0,C 180,E1 -1573.952,E2 -1573.952} C_VEL
LIN {X 0,Y 587.259,Z 357.951,A -85,B 0,C 180,E1 -1576.989,E2 -1576.989} C_VEL
LIN {X 0,Y 587.287,Z 357.949,A -85,B 0,C 180,E1 -1579.743,E2 -1579.743} C_VEL
LIN {X 0,Y 587.297,Z 357.956,A -85,B 0,C 180,E1 -1582.389,E2 -1582.389} C_VEL
LIN {X 0,Y 587.315,Z 357.942,A -85,B 0,C 180,E1 -1585.654,E2 -1585.654} C_VEL
LIN {X 0,Y 587.316,Z 357.952,A -85,B 0,C 180,E1 -1588.23,E2 -1588.23} C_VEL
LIN {X 0,Y 587.324,Z 357.947,A -85,B 0,C 180,E1 -1590.868,E2 -1590.868} C_VEL
LIN {X 0,Y 587.293,Z 357.95,A -85,B 0,C 180,E1 -1593.828,E2 -1593.828} C_VEL
LIN {X 0,Y 587.285,Z 357.955,A -85,B 0,C 180,E1 -1596.74,E2 -1596.74} C_VEL
LIN {X 0,Y 587.287,Z 357.948,A -85,B 0,C 180,E1 -1599.694,E2 -1599.694} C_VEL
LIN {X 0,Y 587.261,Z 357.954,A -85,B 0,C 180,E1 -1601.871,E2 -1601.871} C_VEL
LIN {X 0,Y 587.286,Z 357.954,A -85,B 0,C 180,E1 -1604.736,E2 -1604.736} C_VEL
LIN {X 0,Y 587.26,Z 357.957,A -85,B 0,C 180,E1 -1606.857,E2 -1606.857} C_VEL
LIN {X 0,Y 587.32,Z 357.947,A -85,B 0,C 180,E1 -1608.962,E2 -1608.962} C_VEL
LIN {X 0,Y 587.297,Z 357.947,A -85,B 0,C 180,E1 -1611.744,E2 -1611.744} C_VEL
LIN {X 0,Y 587.33,Z 357.954,A -85,B 0,C 180,E1 -1614.507,E2 -1614.507} C_VEL
LIN {X 0,Y 587.324,Z 357.945,A -85,B 0,C 180,E1 -1617.257,E2 -1617.257} C_VEL
LIN {X 0,Y 587.34,Z 357.944,A -85,B 0,C 180,E1 -1620,E2 -1620} C_VEL
LIN {X 0,Y 587.357,Z 357.948,A -85,B 0,C 180,E1 -1622.743,E2 -1622.743} C_VEL
LIN {X 0,Y 587.304,Z 357.946,A -85,B 0,C 180,E1 -1625.494,E2 -1625.494} C_VEL
LIN {X 0,Y 587.285,Z 357.948,A -85,B 0,C 180,E1 -1627.564,E2 -1627.564} C_VEL
LIN {X 0,Y 587.263,Z 357.952,A -85,B 0,C 180,E1 -1629.645,E2 -1629.645} C_VEL
LIN {X 0,Y 587.299,Z 357.946,A -85,B 0,C 180,E1 -1631.738,E2 -1631.738} C_VEL
LIN {X 0,Y 587.314,Z 357.954,A -85,B 0,C 180,E1 -1634.554,E2 -1634.554} C_VEL
LIN {X 0,Y 587.289,Z 357.949,A -85,B 0,C 180,E1 -1637.408,E2 -1637.408} C_VEL
LIN {X 0,Y 587.277,Z 357.952,A -85,B 0,C 180,E1 -1638.324,E2 -1638.324} C_VEL
LIN {X 0,Y 586.648,Z 358.036,A -85,B 0,C 180,E1 -1638.896,E2 -1638.896} C_VEL
LIN {X 0,Y 583.835,Z 358.385,A -85,B 0,C 180,E1 -1639.825,E2 -1639.825} C_VEL
LIN {X 0,Y 581.422,Z 358.688,A -85,B 0,C 180,E1 -1640.572,E2 -1640.572} C_VEL
LIN {X 0,Y 580.361,Z 358.814,A -85,B 0,C 180,E1 -1641.148,E2 -1641.148} C_VEL
LIN {X 0,Y 580.262,Z 358.824,A -85,B 0,C 180,E1 -1641.343,E2 -1641.343} C_VEL
LIN {X 0,Y 580.238,Z 358.827,A -85,B 0,C 180,E1 -1643.56,E2 -1643.56} C_VEL
LIN {X 0,Y 580.233,Z 358.831,A -85,B 0,C 180,E1 -1646.326,E2 -1646.326} C_VEL
LIN {X 0,Y 580.253,Z 358.827,A -85,B 0,C 180,E1 -1649.305,E2 -1649.305} C_VEL
LIN {X 0,Y 580.27,Z 358.826,A -85,B 0,C 180,E1 -1652.202,E2 -1652.202} C_VEL
LIN {X 0,Y 580.267,Z 358.834,A -85,B 0,C 180,E1 -1654.698,E2 -1654.698} C_VEL
LIN {X 0,Y 580.253,Z 358.824,A -85,B 0,C 180,E1 -1657.272,E2 -1657.272} C_VEL
LIN {X 0,Y 580.264,Z 358.827,A -85,B 0,C 180,E1 -1660.27,E2 -1660.27} C_VEL
LIN {X 0,Y 580.22,Z 358.831,A -85,B 0,C 180,E1 -1663.387,E2 -1663.387} C_VEL
LIN {X 0,Y 580.217,Z 358.833,A -85,B 0,C 180,E1 -1666.339,E2 -1666.339} C_VEL
LIN {X 0,Y 580.245,Z 358.83,A -85,B 0,C 180,E1 -1669.154,E2 -1669.154} C_VEL
LIN {X 0,Y 580.265,Z 358.825,A -85,B 0,C 180,E1 -1671.93,E2 -1671.93} C_VEL
LIN {X 0,Y 580.2,Z 358.837,A -85,B 0,C 180,E1 -1674.451,E2 -1674.451} C_VEL
LIN {X 0,Y 580.235,Z 358.828,A -85,B 0,C 180,E1 -1676.973,E2 -1676.973} C_VEL
LIN {X 0,Y 580.292,Z 359.046,A -85,B 0,C 180,E1 -1679.678,E2 -1679.678} C_VEL
LIN {X 0,Y 582.095,Z 365.236,A -85,B 0,C 180,E1 -1680.378,E2 -1680.378} C_VEL
LIN {X 0,Y 582.368,Z 369.258,A -85,B 0,C 180,E1 -1680.775,E2 -1680.775} C_VEL
LIN {X 0,Y 582.056,Z 394.296,A -85,B 0,C 180,E1 -1683.201,E2 -1683.201} C_VEL
LIN {X 0,Y 581.7,Z 422.771,A -85,B 0,C 180,E1 -1685.937,E2 -1685.937} C_VEL
LIN {X 0,Y 581.347,Z 452.497,A -85,B 0,C 180,E1 -1688.737,E2 -1688.737} C_VEL
LIN {X 0,Y 581.165,Z 473.29,A -85,B 0,C 180,E1 -1690.647,E2 -1690.647} C_VEL
LIN {X 0,Y 581.908,Z 479.249,A -85,B 0,C 180,E1 -1690.768,E2 -1690.768} C_VEL
LIN {X 0,Y 581.518,Z 641.17,A -85,B 0,C 180,E1 -1692.838,E2 -1692.838} C_VEL
LIN {X 0,Y 581.409,Z 656.717,A -85,B 0,C 180,E1 -1693.182,E2 -1693.182} C_VEL
LIN {X 0,Y 581.284,Z 672.057,A -85,B 0,C 180,E1 -1693.675,E2 -1693.675} C_VEL
LIN {X 0,Y 581.108,Z 686.723,A -85,B 0,C 180,E1 -1694.301,E2 -1694.301} C_VEL
LIN {X 0,Y 580.912,Z 700.019,A -85,B 0,C 180,E1 -1695.014,E2 -1695.014} C_VEL
LIN {X 0,Y 580.788,Z 713.367,A -85,B 0,C 180,E1 -1695.891,E2 -1695.891} C_VEL
LIN {X 0,Y 580.59,Z 725.871,A -85,B 0,C 180,E1 -1696.883,E2 -1696.883} C_VEL
LIN {X 0,Y 580.432,Z 737.072,A -85,B 0,C 180,E1 -1697.945,E2 -1697.945} C_VEL
LIN {X 0,Y 580.337,Z 748.122,A -85,B 0,C 180,E1 -1699.202,E2 -1699.202} C_VEL
LIN {X 0,Y 580.238,Z 757,A -85,B 0,C 180,E1 -1700.414,E2 -1700.414} C_VEL
LIN {X 0,Y 580.195,Z 764.498,A -85,B 0,C 180,E1 -1701.643,E2 -1701.643} C_VEL
LIN {X 0,Y 580.137,Z 771.502,A -85,B 0,C 180,E1 -1703.043,E2 -1703.043} C_VEL
LIN {X 0,Y 580.126,Z 777.01,A -85,B 0,C 180,E1 -1704.439,E2 -1704.439} C_VEL
LIN {X 0,Y 580.087,Z 781.177,A -85,B 0,C 180,E1 -1705.832,E2 -1705.832} C_VEL
LIN {X 0,Y 580.038,Z 784.115,A -85,B 0,C 180,E1 -1707.223,E2 -1707.223} C_VEL
LIN {X 0,Y 580.043,Z 785.882,A -85,B 0,C 180,E1 -1708.613,E2 -1708.613} C_VEL
LIN {X 0,Y 580.035,Z 786.496,A -85,B 0,C 180,E1 -1710.001,E2 -1710.001} C_VEL
LIN {X 0,Y 580.045,Z 785.942,A -85,B 0,C 180,E1 -1711.39,E2 -1711.39} C_VEL
LIN {X 0,Y 580.04,Z 784.255,A -85,B 0,C 180,E1 -1712.779,E2 -1712.779} C_VEL
LIN {X 0,Y 580.088,Z 781.401,A -85,B 0,C 180,E1 -1714.17,E2 -1714.17} C_VEL
LIN {X 0,Y 580.123,Z 777.317,A -85,B 0,C 180,E1 -1715.563,E2 -1715.563} C_VEL
LIN {X 0,Y 580.14,Z 771.901,A -85,B 0,C 180,E1 -1716.959,E2 -1716.959} C_VEL
LIN {X 0,Y 580.174,Z 764.997,A -85,B 0,C 180,E1 -1718.359,E2 -1718.359} C_VEL
LIN {X 0,Y 580.235,Z 756.395,A -85,B 0,C 180,E1 -1719.764,E2 -1719.764} C_VEL
LIN {X 0,Y 580.309,Z 746.826,A -85,B 0,C 180,E1 -1721.047,E2 -1721.047} C_VEL
LIN {X 0,Y 580.474,Z 736.191,A -85,B 0,C 180,E1 -1722.233,E2 -1722.233} C_VEL
LIN {X 0,Y 580.607,Z 724.809,A -85,B 0,C 180,E1 -1723.297,E2 -1723.297} C_VEL
LIN {X 0,Y 580.762,Z 712.059,A -85,B 0,C 180,E1 -1724.292,E2 -1724.292} C_VEL
LIN {X 0,Y 580.926,Z 698.456,A -85,B 0,C 180,E1 -1725.167,E2 -1725.167} C_VEL
LIN {X 0,Y 581.119,Z 684.768,A -85,B 0,C 180,E1 -1725.881,E2 -1725.881} C_VEL
LIN {X 0,Y 581.267,Z 670.749,A -85,B 0,C 180,E1 -1726.463,E2 -1726.463} C_VEL
LIN {X 0,Y 581.449,Z 655.712,A -85,B 0,C 180,E1 -1726.933,E2 -1726.933} C_VEL
LIN {X 0,Y 581.506,Z 641.26,A -85,B 0,C 180,E1 -1727.251,E2 -1727.251} C_VEL
LIN {X 0,Y 581.832,Z 477.587,A -85,B 0,C 180,E1 -1729.346,E2 -1729.346} C_VEL
LIN {X 0,Y 581.171,Z 473.057,A -85,B 0,C 180,E1 -1729.456,E2 -1729.456} C_VEL
LIN {X 0,Y 581.465,Z 441.535,A -85,B 0,C 180,E1 -1732.38,E2 -1732.38} C_VEL
LIN {X 0,Y 581.826,Z 412.167,A -85,B 0,C 180,E1 -1735.165,E2 -1735.165} C_VEL
LIN {X 0,Y 582.249,Z 382.044,A -85,B 0,C 180,E1 -1738.084,E2 -1738.084} C_VEL
LIN {X 0,Y 582.244,Z 365.834,A -85,B 0,C 180,E1 -1739.648,E2 -1739.648} C_VEL
LIN {X 0,Y 580.254,Z 358.981,A -85,B 0,C 180,E1 -1740.427,E2 -1740.427} C_VEL
LIN {X 0,Y 580.235,Z 358.828,A -85,B 0,C 180,E1 -1743.306,E2 -1743.306} C_VEL
LIN {X 0,Y 580.227,Z 358.83,A -85,B 0,C 180,E1 -1746.407,E2 -1746.407} C_VEL
LIN {X 0,Y 580.259,Z 358.833,A -85,B 0,C 180,E1 -1749.181,E2 -1749.181} C_VEL
LIN {X 0,Y 580.234,Z 358.828,A -85,B 0,C 180,E1 -1751.774,E2 -1751.774} C_VEL
LIN {X 0,Y 580.228,Z 358.831,A -85,B 0,C 180,E1 -1754.631,E2 -1754.631} C_VEL
LIN {X 0,Y 580.248,Z 358.829,A -85,B 0,C 180,E1 -1757.633,E2 -1757.633} C_VEL
LIN {X 0,Y 580.266,Z 358.821,A -85,B 0,C 180,E1 -1760.065,E2 -1760.065} C_VEL
LIN {X 0,Y 580.268,Z 358.833,A -85,B 0,C 180,E1 -1763.071,E2 -1763.071} C_VEL
LIN {X 0,Y 580.257,Z 358.823,A -85,B 0,C 180,E1 -1766.141,E2 -1766.141} C_VEL
LIN {X 0,Y 580.253,Z 358.828,A -85,B 0,C 180,E1 -1768.613,E2 -1768.613} C_VEL
LIN {X 0,Y 580.269,Z 358.832,A -85,B 0,C 180,E1 -1771.023,E2 -1771.023} C_VEL
LIN {X 0,Y 580.252,Z 358.828,A -85,B 0,C 180,E1 -1773.675,E2 -1773.675} C_VEL
LIN {X 0,Y 580.254,Z 358.827,A -85,B 0,C 180,E1 -1776.441,E2 -1776.441} C_VEL
LIN {X 0,Y 580.268,Z 358.833,A -85,B 0,C 180,E1 -1779.437,E2 -1779.437} C_VEL
LIN {X 0,Y 580.306,Z 358.954,A -85,B 0,C 180,E1 -1780.748,E2 -1780.748} C_VEL
LIN {X 0,Y 580.556,Z 363.087,A -85,B 0,C 180,E1 -1781.472,E2 -1781.472} C_VEL
LIN {X 0,Y 580.508,Z 375.343,A -85,B 0,C 180,E1 -1783.471,E2 -1783.471} C_VEL
LIN {X 0,Y 581.067,Z 378.606,A -85,B 0,C 180,E1 -1783.567,E2 -1783.567} C_VEL
LIN {X 0,Y 581.356,Z 382.984,A -85,B 0,C 180,E1 -1783.631,E2 -1783.631} C_VEL
LIN {X 0,Y 581.142,Z 511.915,A -85,B 0,C 180,E1 -1785.265,E2 -1785.265} C_VEL
LIN {X 0,Y 581.072,Z 526.49,A -85,B 0,C 180,E1 -1785.602,E2 -1785.602} C_VEL
LIN {X 0,Y 580.926,Z 540.873,A -85,B 0,C 180,E1 -1786.087,E2 -1786.087} C_VEL
LIN {X 0,Y 580.774,Z 554.536,A -85,B 0,C 180,E1 -1786.708,E2 -1786.708} C_VEL
LIN {X 0,Y 580.665,Z 566.797,A -85,B 0,C 180,E1 -1787.417,E2 -1787.417} C_VEL
LIN {X 0,Y 580.529,Z 579.418,A -85,B 0,C 180,E1 -1788.318,E2 -1788.318} C_VEL
LIN {X 0,Y 580.442,Z 589.423,A -85,B 0,C 180,E1 -1789.188,E2 -1789.188} C_VEL
LIN {X 0,Y 580.28,Z 599.469,A -85,B 0,C 180,E1 -1790.238,E2 -1790.238} C_VEL
LIN {X 0,Y 580.241,Z 607.849,A -85,B 0,C 180,E1 -1791.292,E2 -1791.292} C_VEL
LIN {X 0,Y 580.167,Z 615.878,A -85,B 0,C 180,E1 -1792.517,E2 -1792.517} C_VEL
LIN {X 0,Y 580.103,Z 622.335,A -85,B 0,C 180,E1 -1793.74,E2 -1793.74} C_VEL
LIN {X 0,Y 580.077,Z 626.783,A -85,B 0,C 180,E1 -1794.786,E2 -1794.786} C_VEL
LIN {X 0,Y 580.103,Z 630.32,A -85,B 0,C 180,E1 -1795.831,E2 -1795.831} C_VEL
LIN {X 0,Y 580.042,Z 633.742,A -85,B 0,C 180,E1 -1797.222,E2 -1797.222} C_VEL
LIN {X 0,Y 580.045,Z 635.777,A -85,B 0,C 180,E1 -1798.611,E2 -1798.611} C_VEL
LIN {X 0,Y 580.034,Z 636.496,A -85,B 0,C 180,E1 -1800,E2 -1800} C_VEL
LIN {X 0,Y 580.041,Z 635.88,A -85,B 0,C 180,E1 -1801.389,E2 -1801.389} C_VEL
LIN {X 0,Y 580.041,Z 633.922,A -85,B 0,C 180,E1 -1802.778,E2 -1802.778} C_VEL
LIN {X 0,Y 580.104,Z 630.581,A -85,B 0,C 180,E1 -1804.168,E2 -1804.168} C_VEL
LIN {X 0,Y 580.128,Z 625.765,A -85,B 0,C 180,E1 -1805.562,E2 -1805.562} C_VEL
LIN {X 0,Y 580.143,Z 619.302,A -85,B 0,C 180,E1 -1806.958,E2 -1806.958} C_VEL
LIN {X 0,Y 580.193,Z 612.104,A -85,B 0,C 180,E1 -1808.183,E2 -1808.183} C_VEL
LIN {X 0,Y 580.275,Z 603.169,A -85,B 0,C 180,E1 -1809.41,E2 -1809.41} C_VEL
LIN {X 0,Y 580.356,Z 593.828,A -85,B 0,C 180,E1 -1810.466,E2 -1810.466} C_VEL
LIN {X 0,Y 580.471,Z 583.855,A -85,B 0,C 180,E1 -1811.404,E2 -1811.404} C_VEL
LIN {X 0,Y 580.582,Z 572.103,A -85,B 0,C 180,E1 -1812.319,E2 -1812.319} C_VEL
LIN {X 0,Y 580.72,Z 559.468,A -85,B 0,C 180,E1 -1813.116,E2 -1813.116} C_VEL
LIN {X 0,Y 580.888,Z 546.178,A -85,B 0,C 180,E1 -1813.78,E2 -1813.78} C_VEL
LIN {X 0,Y 581.021,Z 532.846,A -85,B 0,C 180,E1 -1814.293,E2 -1814.293} C_VEL
LIN {X 0,Y 581.095,Z 519.351,A -85,B 0,C 180,E1 -1814.672,E2 -1814.672} C_VEL
LIN {X 0,Y 581.169,Z 504.62,A -85,B 0,C 180,E1 -1814.935,E2 -1814.935} C_VEL
LIN {X 0,Y 581.299,Z 379.844,A -85,B 0,C 180,E1 -1816.5,E2 -1816.5} C_VEL
LIN {X 0,Y 580.495,Z 375.642,A -85,B 0,C 180,E1 -1816.598,E2 -1816.598} C_VEL
LIN {X 0,Y 580.421,Z 373.18,A -85,B 0,C 180,E1 -1816.947,E2 -1816.947} C_VEL
LIN {X 0,Y 580.508,Z 360.337,A -85,B 0,C 180,E1 -1819.079,E2 -1819.079} C_VEL
LIN {X 0,Y 580.309,Z 358.901,A -85,B 0,C 180,E1 -1819.367,E2 -1819.367} C_VEL
LIN {X 0,Y 580.27,Z 358.827,A -85,B 0,C 180,E1 -1822.053,E2 -1822.053} C_VEL
LIN {X 0,Y 580.311,Z 358.825,A -85,B 0,C 180,E1 -1825.079,E2 -1825.079} C_VEL
LIN {X 0,Y 580.3,Z 358.823,A -85,B 0,C 180,E1 -1828.185,E2 -1828.185} C_VEL
LIN {X 0,Y 580.286,Z 358.831,A -85,B 0,C 180,E1 -1830.694,E2 -1830.694} C_VEL
LIN {X 0,Y 580.306,Z 358.821,A -85,B 0,C 180,E1 -1833.316,E2 -1833.316} C_VEL
LIN {X 0,Y 580.249,Z 358.828,A -85,B 0,C 180,E1 -1835.756,E2 -1835.756} C_VEL
LIN {X 0,Y 580.288,Z 358.828,A -85,B 0,C 180,E1 -1838.146,E2 -1838.146} C_VEL
LIN {X 0,Y 580.296,Z 358.824,A -85,B 0,C 180,E1 -1840.844,E2 -1840.844} C_VEL
LIN {X 0,Y 580.244,Z 358.829,A -85,B 0,C 180,E1 -1843.661,E2 -1843.661} C_VEL
LIN {X 0,Y 580.238,Z 358.832,A -85,B 0,C 180,E1 -1846.613,E2 -1846.613} C_VEL
LIN {X 0,Y 580.278,Z 358.824,A -85,B 0,C 180,E1 -1849.154,E2 -1849.154} C_VEL
LIN {X 0,Y 580.281,Z 358.832,A -85,B 0,C 180,E1 -1851.928,E2 -1851.928} C_VEL
LIN {X 0,Y 580.219,Z 358.834,A -85,B 0,C 180,E1 -1854.45,E2 -1854.45} C_VEL
LIN {X 0,Y 580.241,Z 358.829,A -85,B 0,C 180,E1 -1856.971,E2 -1856.971} C_VEL
LIN {X 0,Y 580.268,Z 358.831,A -85,B 0,C 180,E1 -1859.423,E2 -1859.423} C_VEL
LIN {X 0,Y 580.29,Z 359.051,A -85,B 0,C 180,E1 -1860.547,E2 -1860.547} C_VEL
LIN {X 0,Y 582.486,Z 366.794,A -85,B 0,C 180,E1 -1861.337,E2 -1861.337} C_VEL
LIN {X 0,Y 582.067,Z 396.986,A -85,B 0,C 180,E1 -1864.043,E2 -1864.043} C_VEL
LIN {X 0,Y 581.675,Z 429.552,A -85,B 0,C 180,E1 -1866.904,E2 -1866.904} C_VEL
LIN {X 0,Y 581.296,Z 462.591,A -85,B 0,C 180,E1 -1869.751,E2 -1869.751} C_VEL
LIN {X 0,Y 581.26,Z 473.019,A -85,B 0,C 180,E1 -1870.613,E2 -1870.613} C_VEL
LIN {X 0,Y 581.896,Z 478.384,A -85,B 0,C 180,E1 -1870.711,E2 -1870.711} C_VEL
LIN {X 0,Y 581.539,Z 641.315,A -85,B 0,C 180,E1 -1872.795,E2 -1872.795} C_VEL
LIN {X 0,Y 581.411,Z 656.683,A -85,B 0,C 180,E1 -1873.135,E2 -1873.135} C_VEL
LIN {X 0,Y 581.247,Z 672.025,A -85,B 0,C 180,E1 -1873.627,E2 -1873.627} C_VEL
LIN {X 0,Y 581.126,Z 685.743,A -85,B 0,C 180,E1 -1874.209,E2 -1874.209} C_VEL
LIN {X 0,Y 580.945,Z 699.223,A -85,B 0,C 180,E1 -1874.923,E2 -1874.923} C_VEL
LIN {X 0,Y 580.798,Z 712.47,A -85,B 0,C 180,E1 -1875.782,E2 -1875.782} C_VEL
LIN {X 0,Y 580.609,Z 724.279,A -85,B 0,C 180,E1 -1876.703,E2 -1876.703} C_VEL
LIN {X 0,Y 580.48,Z 735.739,A -85,B 0,C 180,E1 -1877.767,E2 -1877.767} C_VEL
LIN {X 0,Y 580.308,Z 746.453,A -85,B 0,C 180,E1 -1878.953,E2 -1878.953} C_VEL
LIN {X 0,Y 580.268,Z 754.849,A -85,B 0,C 180,E1 -1880.061,E2 -1880.061} C_VEL
LIN {X 0,Y 580.214,Z 762.724,A -85,B 0,C 180,E1 -1881.29,E2 -1881.29} C_VEL
LIN {X 0,Y 580.132,Z 770.083,A -85,B 0,C 180,E1 -1882.691,E2 -1882.691} C_VEL
LIN {X 0,Y 580.129,Z 775.921,A -85,B 0,C 180,E1 -1884.089,E2 -1884.089} C_VEL
LIN {X 0,Y 580.041,Z 779.381,A -85,B 0,C 180,E1 -1885.134,E2 -1885.134} C_VEL
LIN {X 0,Y 580.105,Z 782.884,A -85,B 0,C 180,E1 -1886.526,E2 -1886.526} C_VEL
LIN {X 0,Y 580.036,Z 785.191,A -85,B 0,C 180,E1 -1887.916,E2 -1887.916} C_VEL
LIN {X 0,Y 580.038,Z 786.349,A -85,B 0,C 180,E1 -1889.305,E2 -1889.305} C_VEL
LIN {X 0,Y 580.038,Z 786.35,A -85,B 0,C 180,E1 -1890.693,E2 -1890.693} C_VEL
LIN {X 0,Y 580.036,Z 785.194,A -85,B 0,C 180,E1 -1892.082,E2 -1892.082} C_VEL
LIN {X 0,Y 580.105,Z 782.89,A -85,B 0,C 180,E1 -1893.472,E2 -1893.472} C_VEL
LIN {X 0,Y 580.041,Z 779.388,A -85,B 0,C 180,E1 -1894.864,E2 -1894.864} C_VEL
LIN {X 0,Y 580.091,Z 774.612,A -85,B 0,C 180,E1 -1896.259,E2 -1896.259} C_VEL
LIN {X 0,Y 580.168,Z 768.431,A -85,B 0,C 180,E1 -1897.656,E2 -1897.656} C_VEL
LIN {X 0,Y 580.207,Z 760.66,A -85,B 0,C 180,E1 -1899.059,E2 -1899.059} C_VEL
LIN {X 0,Y 580.308,Z 752.379,A -85,B 0,C 180,E1 -1900.289,E2 -1900.289} C_VEL
LIN {X 0,Y 580.381,Z 742.406,A -85,B 0,C 180,E1 -1901.524,E2 -1901.524} C_VEL
LIN {X 0,Y 580.54,Z 732.203,A -85,B 0,C 180,E1 -1902.585,E2 -1902.585} C_VEL
LIN {X 0,Y 580.677,Z 720.031,A -85,B 0,C 180,E1 -1903.65,E2 -1903.65} C_VEL
LIN {X 0,Y 580.871,Z 706.543,A -85,B 0,C 180,E1 -1904.624,E2 -1904.624} C_VEL
LIN {X 0,Y 581.016,Z 692.896,A -85,B 0,C 180,E1 -1905.432,E2 -1905.432} C_VEL
LIN {X 0,Y 581.208,Z 678.829,A -85,B 0,C 180,E1 -1906.101,E2 -1906.101} C_VEL
LIN {X 0,Y 581.348,Z 664.336,A -85,B 0,C 180,E1 -1906.639,E2 -1906.639} C_VEL
LIN {X 0,Y 581.496,Z 649.028,A -85,B 0,C 180,E1 -1907.053,E2 -1907.053} C_VEL
LIN {X 0,Y 581.554,Z 633.526,A -85,B 0,C 180,E1 -1907.323,E2 -1907.323} C_VEL
LIN {X 0,Y 581.805,Z 476.649,A -85,B 0,C 180,E1 -1909.314,E2 -1909.314} C_VEL
LIN {X 0,Y 581.228,Z 472.504,A -85,B 0,C 180,E1 -1909.413,E2 -1909.413} C_VEL
LIN {X 0,Y 581.572,Z 437.882,A -85,B 0,C 180,E1 -1912.373,E2 -1912.373} C_VEL
LIN {X 0,Y 581.971,Z 404.652,A -85,B 0,C 180,E1 -1915.278,E2 -1915.278} C_VEL
LIN {X 0,Y 582.427,Z 373.352,A -85,B 0,C 180,E1 -1918.072,E2 -1918.072} C_VEL
LIN {X 0,Y 582.486,Z 366.814,A -85,B 0,C 180,E1 -1918.661,E2 -1918.661} C_VEL
LIN {X 0,Y 580.27,Z 359.023,A -85,B 0,C 180,E1 -1919.486,E2 -1919.486} C_VEL
LIN {X 0,Y 580.275,Z 358.83,A -85,B 0,C 180,E1 -1922.026,E2 -1922.026} C_VEL
LIN {X 0,Y 580.26,Z 358.829,A -85,B 0,C 180,E1 -1924.696,E2 -1924.696} C_VEL
LIN {X 0,Y 580.255,Z 358.826,A -85,B 0,C 180,E1 -1927.27,E2 -1927.27} C_VEL
LIN {X 0,Y 580.269,Z 358.834,A -85,B 0,C 180,E1 -1930.268,E2 -1930.268} C_VEL
LIN {X 0,Y 580.258,Z 358.829,A -85,B 0,C 180,E1 -1932.706,E2 -1932.706} C_VEL
LIN {X 0,Y 580.223,Z 358.83,A -85,B 0,C 180,E1 -1935.612,E2 -1935.612} C_VEL
LIN {X 0,Y 580.226,Z 358.832,A -85,B 0,C 180,E1 -1938.227,E2 -1938.227} C_VEL
LIN {X 0,Y 580.246,Z 358.828,A -85,B 0,C 180,E1 -1940.963,E2 -1940.963} C_VEL
LIN {X 0,Y 580.223,Z 358.827,A -85,B 0,C 180,E1 -1943.593,E2 -1943.593} C_VEL
LIN {X 0,Y 580.262,Z 358.825,A -85,B 0,C 180,E1 -1946.142,E2 -1946.142} C_VEL
LIN {X 0,Y 580.25,Z 358.832,A -85,B 0,C 180,E1 -1948.613,E2 -1948.613} C_VEL
LIN {X 0,Y 580.261,Z 358.825,A -85,B 0,C 180,E1 -1951.022,E2 -1951.022} C_VEL
LIN {X 0,Y 580.25,Z 358.831,A -85,B 0,C 180,E1 -1954.149,E2 -1954.149} C_VEL
LIN {X 0,Y 580.261,Z 358.825,A -85,B 0,C 180,E1 -1957.196,E2 -1957.196} C_VEL
LIN {X 0,Y 580.256,Z 358.829,A -85,B 0,C 180,E1 -1960.176,E2 -1960.176} C_VEL
LIN {X 0,Y 580.211,Z 358.832,A -85,B 0,C 180,E1 -1963.114,E2 -1963.114} C_VEL
